KUKA KRL program: f1_Kuka_APT215T03S15.SRC

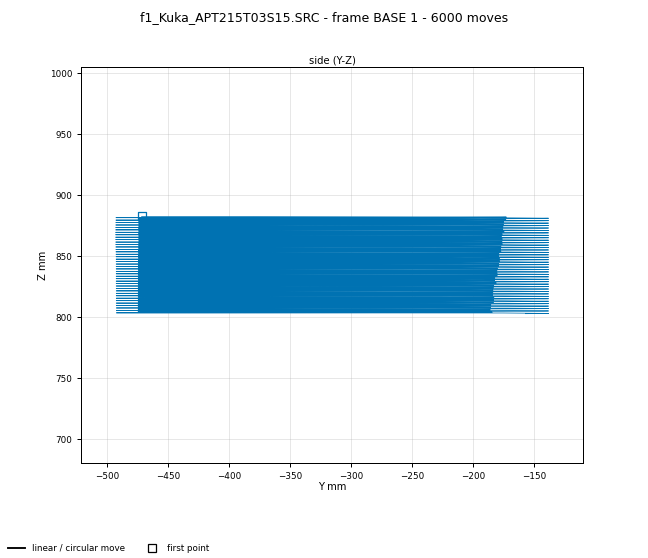
[picture p0: tool path of f1_Kuka_APT215T03S15.SRC in frame BASE 1, 6000 of 6001 moves have a stored position in this frame; points joined in program order, loops and branches not executed]
&ACCESS RVP
&REL 2
&PARAM TEMPLATE = C:\KRC\Roboter\Template\vorgabe
&PARAM EDITMASK = *
DEF f1_Kuka_APT215T03S15()


;FOLD INI;%{PE}%V3.2.0,%MKUKATPBASIS,%CINIT,%VCOMMON,%P
  ;FOLD BAS INI;%{E}%V3.2.0,%MKUKATPBASIS,%CINIT,%VINIT,%P
    GLOBAL INTERRUPT DECL 3 WHEN $STOPMESS==TRUE DO IR_STOPM ( )
    INTERRUPT ON 3
    BAS (#INITMOV,0 )
  ;ENDFOLD (BAS INI)
  ;FOLD USER INI;%{E}%V3.2.0,%MKUKATPUSER,%CINIT,%VINIT,%P
    ;Make your modifications here
  ;ENDFOLD (USER INI)
;ENDFOLD (INI)


;*** Make Null PTP Move
  PTP $pos_act

;*** Auto Load The Correct TOOL Data
  $tool=tool_data[3]

;*** Auto Load The Correct BASE Data
  $base=base_data[1]

  $ADVANCE = 5

;*** Restate Last Velocity
MMPM(30000.0)
SetRPM(6000)
LIN {X 0.010,Y -471.850,Z 882.542,A 0.000,B 0.000,C 90.000,E1 97.466} C_DIS
LIN {X -0.193,Y -470.473,Z 882.540,A 0.000,B 0.000,C 90.000,E1 97.239} C_DIS
LIN {X -0.077,Y -455.997,Z 882.527,A 0.000,B 0.000,C 90.000,E1 94.935} C_DIS
LIN {X -0.109,Y -443.986,Z 882.516,A 0.000,B 0.000,C 90.000,E1 92.865} C_DIS
LIN {X -0.078,Y -436.155,Z 882.509,A 0.000,B 0.000,C 90.000,E1 91.547} C_DIS
LIN {X -0.026,Y -426.626,Z 882.500,A 0.000,B 0.000,C 90.000,E1 89.943} C_DIS
LIN {X -0.024,Y -415.186,Z 882.489,A 0.000,B 0.000,C 90.000,E1 88.051} C_DIS
LIN {X 0.145,Y -403.849,Z 882.478,A 0.000,B 0.000,C 90.000,E1 86.102} C_DIS
LIN {X 0.181,Y -390.966,Z 882.466,A 0.000,B 0.000,C 90.000,E1 83.856} C_DIS
LIN {X -0.053,Y -379.852,Z 882.455,A 0.000,B 0.000,C 90.000,E1 81.894} C_DIS
LIN {X -0.034,Y -368.671,Z 882.444,A 0.000,B 0.000,C 90.000,E1 79.859} C_DIS
LIN {X 0.178,Y -357.598,Z 882.432,A 0.000,B 0.000,C 90.000,E1 77.757} C_DIS
LIN {X -0.125,Y -346.414,Z 882.420,A 0.000,B 0.000,C 90.000,E1 75.700} C_DIS
LIN {X 0.159,Y -333.850,Z 882.407,A 0.000,B 0.000,C 90.000,E1 73.196} C_DIS
LIN {X -0.086,Y -321.740,Z 882.393,A 0.000,B 0.000,C 90.000,E1 70.732} C_DIS
LIN {X 0.000,Y -309.964,Z 882.379,A 0.000,B 0.000,C 90.000,E1 68.156} C_DIS
LIN {X 0.018,Y -299.904,Z 882.366,A 0.000,B 0.000,C 90.000,E1 65.869} C_DIS
LIN {X -0.085,Y -289.792,Z 882.353,A 0.000,B 0.000,C 90.000,E1 63.563} C_DIS
LIN {X -0.007,Y -279.667,Z 882.340,A 0.000,B 0.000,C 90.000,E1 61.179} C_DIS
LIN {X 0.035,Y -268.308,Z 882.325,A 0.000,B 0.000,C 90.000,E1 58.408} C_DIS
LIN {X -0.117,Y -256.237,Z 882.307,A 0.000,B 0.000,C 90.000,E1 55.261} C_DIS
LIN {X -0.007,Y -245.352,Z 882.289,A 0.000,B 0.000,C 90.000,E1 51.984} C_DIS
LIN {X 0.087,Y -236.617,Z 882.272,A 0.000,B 0.000,C 90.000,E1 49.013} C_DIS
LIN {X -0.003,Y -226.592,Z 882.252,A 0.000,B 0.000,C 90.000,E1 45.283} C_DIS
LIN {X -0.070,Y -217.235,Z 882.230,A 0.000,B 0.000,C 90.000,E1 41.472} C_DIS
LIN {X 0.094,Y -208.562,Z 882.209,A 0.000,B 0.000,C 90.000,E1 37.523} C_DIS
LIN {X -0.113,Y -202.133,Z 882.191,A 0.000,B 0.000,C 90.000,E1 34.405} C_DIS
LIN {X 0.076,Y -196.229,Z 882.173,A 0.000,B 0.000,C 90.000,E1 31.131} C_DIS
LIN {X -0.021,Y -190.898,Z 882.155,A 0.000,B 0.000,C 90.000,E1 27.897} C_DIS
LIN {X -0.002,Y -186.219,Z 882.137,A 0.000,B 0.000,C 90.000,E1 24.591} C_DIS
LIN {X -0.079,Y -182.268,Z 882.118,A 0.000,B 0.000,C 90.000,E1 21.280} C_DIS
LIN {X 0.019,Y -178.306,Z 882.095,A 0.000,B 0.000,C 90.000,E1 17.040} C_DIS
LIN {X -0.012,Y -175.022,Z 882.066,A 0.000,B 0.000,C 90.000,E1 11.951} C_DIS
LIN {X -0.015,Y -172.998,Z 882.024,A 0.000,B 0.000,C 90.000,E1 4.245} C_DIS
LIN {X 0.007,Y -174.503,Z 881.974,A 0.000,B 0.000,C 90.000,E1 355.241} C_DIS
LIN {X 0.070,Y -177.369,Z 881.945,A 0.000,B 0.000,C 90.000,E1 350.095} C_DIS
LIN {X -0.017,Y -180.888,Z 881.922,A 0.000,B 0.000,C 90.000,E1 345.880} C_DIS
LIN {X 0.057,Y -184.611,Z 881.903,A 0.000,B 0.000,C 90.000,E1 342.489} C_DIS
LIN {X 0.038,Y -189.077,Z 881.884,A 0.000,B 0.000,C 90.000,E1 339.156} C_DIS
LIN {X -0.021,Y -194.301,Z 881.866,A 0.000,B 0.000,C 90.000,E1 335.869} C_DIS
LIN {X 0.062,Y -201.598,Z 881.843,A 0.000,B 0.000,C 90.000,E1 331.769} C_DIS
LIN {X -0.041,Y -209.434,Z 881.821,A 0.000,B 0.000,C 90.000,E1 327.788} C_DIS
LIN {X 0.024,Y -218.033,Z 881.799,A 0.000,B 0.000,C 90.000,E1 323.829} C_DIS
LIN {X 0.049,Y -225.580,Z 881.782,A 0.000,B 0.000,C 90.000,E1 320.723} C_DIS
LIN {X 0.044,Y -233.817,Z 881.765,A 0.000,B 0.000,C 90.000,E1 317.676} C_DIS
LIN {X 0.081,Y -243.078,Z 881.748,A 0.000,B 0.000,C 90.000,E1 314.676} C_DIS
LIN {X 0.028,Y -254.595,Z 881.730,A 0.000,B 0.000,C 90.000,E1 311.391} C_DIS
LIN {X -0.008,Y -267.268,Z 881.712,A 0.000,B 0.000,C 90.000,E1 308.177} C_DIS
LIN {X 0.040,Y -281.099,Z 881.695,A 0.000,B 0.000,C 90.000,E1 305.025} C_DIS
LIN {X -0.167,Y -296.298,Z 881.678,A 0.000,B 0.000,C 90.000,E1 302.005} C_DIS
LIN {X -0.039,Y -311.051,Z 881.663,A 0.000,B 0.000,C 90.000,E1 299.333} C_DIS
LIN {X 0.005,Y -323.057,Z 881.652,A 0.000,B 0.000,C 90.000,E1 297.385} C_DIS
LIN {X 0.118,Y -338.511,Z 881.640,A 0.000,B 0.000,C 90.000,E1 295.155} C_DIS
LIN {X 0.107,Y -357.539,Z 881.626,A 0.000,B 0.000,C 90.000,E1 292.717} C_DIS
LIN {X 0.020,Y -380.471,Z 881.612,A 0.000,B 0.000,C 90.000,E1 290.066} C_DIS
LIN {X -0.081,Y -403.987,Z 881.598,A 0.000,B 0.000,C 90.000,E1 287.583} C_DIS
LIN {X -0.193,Y -416.845,Z 881.590,A 0.000,B 0.000,C 90.000,E1 286.260} C_DIS
LIN {X -0.043,Y -429.200,Z 881.583,A 0.000,B 0.000,C 90.000,E1 284.898} C_DIS
LIN {X -0.037,Y -438.799,Z 881.577,A 0.000,B 0.000,C 90.000,E1 283.828} C_DIS
LIN {X 0.178,Y -450.162,Z 881.569,A 0.000,B 0.000,C 90.000,E1 282.479} C_DIS
LIN {X 0.044,Y -456.611,Z 881.565,A 0.000,B 0.000,C 90.000,E1 281.715} C_DIS
LIN {X 0.242,Y -464.630,Z 881.559,A 0.000,B 0.000,C 90.000,E1 280.658} C_DIS
LIN {X -0.013,Y -472.017,Z 881.554,A 0.000,B 0.000,C 90.000,E1 279.670} C_DIS
LIN {X -0.192,Y -478.710,Z 881.548,A 0.000,B 0.000,C 90.000,E1 278.681} C_DIS
LIN {X -0.246,Y -482.946,Z 881.544,A 0.000,B 0.000,C 90.000,E1 277.936} C_DIS
LIN {X -0.189,Y -486.486,Z 881.540,A 0.000,B 0.000,C 90.000,E1 277.182} C_DIS
LIN {X -0.107,Y -489.356,Z 881.536,A 0.000,B 0.000,C 90.000,E1 276.429} C_DIS
LIN {X 0.102,Y -490.795,Z 881.533,A 0.000,B 0.000,C 90.000,E1 275.910} C_DIS
LIN {X -0.169,Y -491.904,Z 881.530,A 0.000,B 0.000,C 90.000,E1 275.448} C_DIS
LIN {X 0.014,Y -492.581,Z 881.527,A 0.000,B 0.000,C 90.000,E1 274.935} C_DIS
LIN {X -0.244,Y -492.872,Z 881.525,A 0.000,B 0.000,C 90.000,E1 274.473} C_DIS
LIN {X -0.009,Y -492.764,Z 881.522,A 0.000,B 0.000,C 90.000,E1 273.955} C_DIS
LIN {X 0.195,Y -492.202,Z 881.519,A 0.000,B 0.000,C 90.000,E1 273.440} C_DIS
LIN {X -0.063,Y -491.234,Z 881.517,A 0.000,B 0.000,C 90.000,E1 272.980} C_DIS
LIN {X 0.140,Y -489.732,Z 881.514,A 0.000,B 0.000,C 90.000,E1 272.465} C_DIS
LIN {X -0.149,Y -487.740,Z 881.511,A 0.000,B 0.000,C 90.000,E1 272.007} C_DIS
LIN {X 0.058,Y -485.217,Z 881.508,A 0.000,B 0.000,C 90.000,E1 271.489} C_DIS
LIN {X 0.229,Y -481.976,Z 881.506,A 0.000,B 0.000,C 90.000,E1 270.974} C_DIS
LIN {X -0.096,Y -477.977,Z 881.503,A 0.000,B 0.000,C 90.000,E1 270.516} C_DIS
LIN {X 0.039,Y -473.005,Z 881.500,A 0.000,B 0.000,C 90.000,E1 270.000} C_DIS
LIN {X -0.168,Y -467.225,Z 881.497,A 0.000,B 0.000,C 90.000,E1 269.542} C_DIS
LIN {X 0.073,Y -461.050,Z 881.495,A 0.000,B 0.000,C 90.000,E1 269.083} C_DIS
LIN {X -0.184,Y -454.316,Z 881.493,A 0.000,B 0.000,C 90.000,E1 268.740} C_DIS
LIN {X 0.053,Y -447.342,Z 881.491,A 0.000,B 0.000,C 90.000,E1 268.396} C_DIS
LIN {X -0.151,Y -439.936,Z 881.490,A 0.000,B 0.000,C 90.000,E1 268.165} C_DIS
LIN {X 0.051,Y -432.196,Z 881.489,A 0.000,B 0.000,C 90.000,E1 267.936} C_DIS
LIN {X 0.202,Y -424.431,Z 881.488,A 0.000,B 0.000,C 90.000,E1 267.764} C_DIS
LIN {X -0.029,Y -417.358,Z 881.487,A 0.000,B 0.000,C 90.000,E1 267.707} C_DIS
LIN {X 0.050,Y -409.094,Z 881.487,A 0.000,B 0.000,C 90.000,E1 267.650} C_DIS
LIN {X -0.005,Y -181.071,Z 881.487,A 0.000,B 0.000,C 90.000,E1 267.650} C_DIS
LIN {X 0.042,Y -180.878,Z 881.473,A 0.000,B 0.000,C 90.000,E1 265.065} C_DIS
LIN {X -0.078,Y -178.996,Z 881.445,A 0.000,B 0.000,C 90.000,E1 260.038} C_DIS
LIN {X 0.016,Y -178.582,Z 881.440,A 0.000,B 0.000,C 90.000,E1 259.162} C_DIS
LIN {X -0.090,Y -175.636,Z 881.411,A 0.000,B 0.000,C 90.000,E1 254.102} C_DIS
LIN {X -0.024,Y -172.355,Z 881.388,A 0.000,B 0.000,C 90.000,E1 249.806} C_DIS
LIN {X -0.069,Y -171.140,Z 881.378,A 0.000,B 0.000,C 90.000,E1 248.103} C_DIS
LIN {X -0.024,Y -167.444,Z 881.354,A 0.000,B 0.000,C 90.000,E1 243.768} C_DIS
LIN {X 0.058,Y -166.840,Z 881.349,A 0.000,B 0.000,C 90.000,E1 242.871} C_DIS
LIN {X -0.025,Y -162.823,Z 881.325,A 0.000,B 0.000,C 90.000,E1 238.535} C_DIS
LIN {X 0.039,Y -161.509,Z 881.315,A 0.000,B 0.000,C 90.000,E1 236.755} C_DIS
LIN {X -0.008,Y -157.507,Z 881.291,A 0.000,B 0.000,C 90.000,E1 232.351} C_DIS
LIN {X 0.026,Y -155.529,Z 881.276,A 0.000,B 0.000,C 90.000,E1 229.666} C_DIS
LIN {X 0.075,Y -151.826,Z 881.251,A 0.000,B 0.000,C 90.000,E1 225.162} C_DIS
LIN {X 0.087,Y -150.040,Z 881.236,A 0.000,B 0.000,C 90.000,E1 222.447} C_DIS
LIN {X 0.001,Y -146.857,Z 881.211,A 0.000,B 0.000,C 90.000,E1 217.935} C_DIS
LIN {X 0.019,Y -145.441,Z 881.195,A 0.000,B 0.000,C 90.000,E1 215.185} C_DIS
LIN {X 0.014,Y -142.862,Z 881.170,A 0.000,B 0.000,C 90.000,E1 210.590} C_DIS
LIN {X 0.066,Y -141.478,Z 881.149,A 0.000,B 0.000,C 90.000,E1 206.873} C_DIS
LIN {X -0.074,Y -139.380,Z 881.113,A 0.000,B 0.000,C 90.000,E1 200.429} C_DIS
LIN {X 0.047,Y -138.834,Z 881.098,A 0.000,B 0.000,C 90.000,E1 197.583} C_DIS
LIN {X -0.025,Y -138.354,Z 881.056,A 0.000,B 0.000,C 90.000,E1 190.141} C_DIS
LIN {X -0.030,Y -139.524,Z 881.004,A 0.000,B 0.000,C 90.000,E1 180.802} C_DIS
LIN {X 0.063,Y -141.193,Z 880.973,A 0.000,B 0.000,C 90.000,E1 175.179} C_DIS
LIN {X 0.022,Y -142.570,Z 880.958,A 0.000,B 0.000,C 90.000,E1 172.413} C_DIS
LIN {X -0.023,Y -144.858,Z 880.932,A 0.000,B 0.000,C 90.000,E1 167.813} C_DIS
LIN {X -0.068,Y -147.484,Z 880.912,A 0.000,B 0.000,C 90.000,E1 164.157} C_DIS
LIN {X -0.042,Y -150.071,Z 880.892,A 0.000,B 0.000,C 90.000,E1 160.496} C_DIS
LIN {X -0.039,Y -153.420,Z 880.871,A 0.000,B 0.000,C 90.000,E1 156.869} C_DIS
LIN {X 0.010,Y -156.840,Z 880.851,A 0.000,B 0.000,C 90.000,E1 153.256} C_DIS
LIN {X 0.081,Y -160.920,Z 880.832,A 0.000,B 0.000,C 90.000,E1 149.665} C_DIS
LIN {X 0.026,Y -163.045,Z 880.822,A 0.000,B 0.000,C 90.000,E1 147.916} C_DIS
LIN {X 0.030,Y -167.437,Z 880.802,A 0.000,B 0.000,C 90.000,E1 144.402} C_DIS
LIN {X -0.060,Y -171.275,Z 880.788,A 0.000,B 0.000,C 90.000,E1 141.823} C_DIS
LIN {X -0.022,Y -176.168,Z 880.769,A 0.000,B 0.000,C 90.000,E1 138.366} C_DIS
LIN {X -0.024,Y -180.440,Z 880.754,A 0.000,B 0.000,C 90.000,E1 135.810} C_DIS
LIN {X -0.048,Y -185.845,Z 880.736,A 0.000,B 0.000,C 90.000,E1 132.447} C_DIS
LIN {X 0.005,Y -190.467,Z 880.722,A 0.000,B 0.000,C 90.000,E1 129.930} C_DIS
LIN {X -0.053,Y -193.245,Z 880.713,A 0.000,B 0.000,C 90.000,E1 128.302} C_DIS
LIN {X 0.114,Y -294.589,Z 880.713,A 0.000,B 0.000,C 90.000,E1 128.257} C_DIS
LIN {X -0.011,Y -298.435,Z 880.712,A 0.000,B 0.000,C 90.000,E1 128.177} C_DIS
LIN {X 0.067,Y -301.502,Z 880.711,A 0.000,B 0.000,C 90.000,E1 127.971} C_DIS
LIN {X 0.003,Y -305.177,Z 880.709,A 0.000,B 0.000,C 90.000,E1 127.604} C_DIS
LIN {X -0.028,Y -308.676,Z 880.706,A 0.000,B 0.000,C 90.000,E1 127.030} C_DIS
LIN {X -0.066,Y -310.063,Z 880.704,A 0.000,B 0.000,C 90.000,E1 126.710} C_DIS
LIN {X -0.025,Y -313.058,Z 880.698,A 0.000,B 0.000,C 90.000,E1 125.724} C_DIS
LIN {X 0.026,Y -323.493,Z 880.681,A 0.000,B 0.000,C 90.000,E1 122.498} C_DIS
LIN {X -0.040,Y -334.226,Z 880.665,A 0.000,B 0.000,C 90.000,E1 119.667} C_DIS
LIN {X -0.012,Y -346.336,Z 880.649,A 0.000,B 0.000,C 90.000,E1 116.873} C_DIS
LIN {X 0.053,Y -359.926,Z 880.634,A 0.000,B 0.000,C 90.000,E1 114.131} C_DIS
LIN {X -0.037,Y -373.349,Z 880.621,A 0.000,B 0.000,C 90.000,E1 111.770} C_DIS
LIN {X -0.066,Y -388.134,Z 880.608,A 0.000,B 0.000,C 90.000,E1 109.450} C_DIS
LIN {X 0.029,Y -404.388,Z 880.595,A 0.000,B 0.000,C 90.000,E1 107.166} C_DIS
LIN {X 0.029,Y -422.226,Z 880.583,A 0.000,B 0.000,C 90.000,E1 104.954} C_DIS
LIN {X -0.091,Y -441.673,Z 880.571,A 0.000,B 0.000,C 90.000,E1 102.827} C_DIS
LIN {X -0.072,Y -461.927,Z 880.560,A 0.000,B 0.000,C 90.000,E1 100.838} C_DIS
LIN {X -0.063,Y -467.060,Z 880.558,A 0.000,B 0.000,C 90.000,E1 100.366} C_DIS
LIN {X -0.122,Y -469.152,Z 880.556,A 0.000,B 0.000,C 90.000,E1 100.141} C_DIS
LIN {X 0.189,Y -470.867,Z 880.555,A 0.000,B 0.000,C 90.000,E1 99.849} C_DIS
LIN {X 0.037,Y -472.156,Z 880.553,A 0.000,B 0.000,C 90.000,E1 99.613} C_DIS
LIN {X 0.140,Y -473.756,Z 880.551,A 0.000,B 0.000,C 90.000,E1 99.095} C_DIS
LIN {X -0.144,Y -474.301,Z 880.548,A 0.000,B 0.000,C 90.000,E1 98.624} C_DIS
LIN {X -0.022,Y -473.883,Z 880.545,A 0.000,B 0.000,C 90.000,E1 98.106} C_DIS
LIN {X 0.105,Y -472.441,Z 880.542,A 0.000,B 0.000,C 90.000,E1 97.587} C_DIS
LIN {X -0.036,Y -471.263,Z 880.541,A 0.000,B 0.000,C 90.000,E1 97.352} C_DIS
LIN {X 0.122,Y -453.784,Z 880.525,A 0.000,B 0.000,C 90.000,E1 94.531} C_DIS
LIN {X -0.184,Y -443.285,Z 880.515,A 0.000,B 0.000,C 90.000,E1 92.751} C_DIS
LIN {X 0.163,Y -432.309,Z 880.505,A 0.000,B 0.000,C 90.000,E1 90.859} C_DIS
LIN {X 0.015,Y -424.286,Z 880.497,A 0.000,B 0.000,C 90.000,E1 89.542} C_DIS
LIN {X 0.054,Y -411.223,Z 880.485,A 0.000,B 0.000,C 90.000,E1 87.364} C_DIS
LIN {X -0.162,Y -398.253,Z 880.473,A 0.000,B 0.000,C 90.000,E1 85.179} C_DIS
LIN {X 0.146,Y -385.479,Z 880.461,A 0.000,B 0.000,C 90.000,E1 82.875} C_DIS
LIN {X -0.146,Y -374.324,Z 880.449,A 0.000,B 0.000,C 90.000,E1 80.905} C_DIS
LIN {X 0.098,Y -361.590,Z 880.436,A 0.000,B 0.000,C 90.000,E1 78.522} C_DIS
LIN {X -0.063,Y -352.080,Z 880.426,A 0.000,B 0.000,C 90.000,E1 76.756} C_DIS
LIN {X -0.144,Y -339.421,Z 880.413,A 0.000,B 0.000,C 90.000,E1 74.338} C_DIS
LIN {X 0.024,Y -325.599,Z 880.397,A 0.000,B 0.000,C 90.000,E1 71.511} C_DIS
LIN {X 0.166,Y -315.230,Z 880.385,A 0.000,B 0.000,C 90.000,E1 69.263} C_DIS
LIN {X 0.096,Y -302.213,Z 880.369,A 0.000,B 0.000,C 90.000,E1 66.357} C_DIS
LIN {X -0.080,Y -292.138,Z 880.356,A 0.000,B 0.000,C 90.000,E1 64.076} C_DIS
LIN {X 0.047,Y -282.052,Z 880.343,A 0.000,B 0.000,C 90.000,E1 61.691} C_DIS
LIN {X 0.014,Y -270.690,Z 880.328,A 0.000,B 0.000,C 90.000,E1 58.948} C_DIS
LIN {X -0.027,Y -257.195,Z 880.308,A 0.000,B 0.000,C 90.000,E1 55.435} C_DIS
LIN {X -0.032,Y -246.268,Z 880.290,A 0.000,B 0.000,C 90.000,E1 52.190} C_DIS
LIN {X 0.050,Y -235.395,Z 880.269,A 0.000,B 0.000,C 90.000,E1 48.485} C_DIS
LIN {X -0.079,Y -225.504,Z 880.249,A 0.000,B 0.000,C 90.000,E1 44.757} C_DIS
LIN {X -0.026,Y -216.257,Z 880.227,A 0.000,B 0.000,C 90.000,E1 40.906} C_DIS
LIN {X -0.127,Y -209.338,Z 880.210,A 0.000,B 0.000,C 90.000,E1 37.810} C_DIS
LIN {X -0.027,Y -202.848,Z 880.192,A 0.000,B 0.000,C 90.000,E1 34.612} C_DIS
LIN {X 0.010,Y -196.935,Z 880.174,A 0.000,B 0.000,C 90.000,E1 31.386} C_DIS
LIN {X -0.071,Y -191.539,Z 880.156,A 0.000,B 0.000,C 90.000,E1 28.153} C_DIS
LIN {X 0.043,Y -186.802,Z 880.138,A 0.000,B 0.000,C 90.000,E1 24.823} C_DIS
LIN {X -0.095,Y -182.794,Z 880.119,A 0.000,B 0.000,C 90.000,E1 21.535} C_DIS
LIN {X 0.080,Y -178.782,Z 880.096,A 0.000,B 0.000,C 90.000,E1 17.275} C_DIS
LIN {X 0.063,Y -175.424,Z 880.068,A 0.000,B 0.000,C 90.000,E1 12.187} C_DIS
LIN {X -0.071,Y -173.297,Z 880.025,A 0.000,B 0.000,C 90.000,E1 4.531} C_DIS
LIN {X 0.017,Y -174.836,Z 879.974,A 0.000,B 0.000,C 90.000,E1 355.241} C_DIS
LIN {X 0.093,Y -177.721,Z 879.945,A 0.000,B 0.000,C 90.000,E1 350.095} C_DIS
LIN {X 0.016,Y -181.260,Z 879.922,A 0.000,B 0.000,C 90.000,E1 345.880} C_DIS
LIN {X -0.029,Y -186.033,Z 879.898,A 0.000,B 0.000,C 90.000,E1 341.692} C_DIS
LIN {X 0.060,Y -190.719,Z 879.880,A 0.000,B 0.000,C 90.000,E1 338.337} C_DIS
LIN {X 0.046,Y -196.088,Z 879.861,A 0.000,B 0.000,C 90.000,E1 335.049} C_DIS
LIN {X 0.006,Y -203.451,Z 879.839,A 0.000,B 0.000,C 90.000,E1 331.001} C_DIS
LIN {X 0.053,Y -209.729,Z 879.821,A 0.000,B 0.000,C 90.000,E1 327.788} C_DIS
LIN {X 0.003,Y -218.309,Z 879.799,A 0.000,B 0.000,C 90.000,E1 323.863} C_DIS
LIN {X -0.150,Y -225.862,Z 879.782,A 0.000,B 0.000,C 90.000,E1 320.803} C_DIS
LIN {X 0.017,Y -234.095,Z 879.765,A 0.000,B 0.000,C 90.000,E1 317.715} C_DIS
LIN {X -0.122,Y -243.332,Z 879.748,A 0.000,B 0.000,C 90.000,E1 314.757} C_DIS
LIN {X -0.008,Y -254.812,Z 879.730,A 0.000,B 0.000,C 90.000,E1 311.434} C_DIS
LIN {X -0.050,Y -267.406,Z 879.712,A 0.000,B 0.000,C 90.000,E1 308.222} C_DIS
LIN {X -0.171,Y -281.188,Z 879.695,A 0.000,B 0.000,C 90.000,E1 305.105} C_DIS
LIN {X 0.037,Y -294.547,Z 879.680,A 0.000,B 0.000,C 90.000,E1 302.339} C_DIS
LIN {X 0.128,Y -309.056,Z 879.665,A 0.000,B 0.000,C 90.000,E1 299.667} C_DIS
LIN {X -0.074,Y -322.902,Z 879.652,A 0.000,B 0.000,C 90.000,E1 297.436} C_DIS
LIN {X 0.026,Y -338.293,Z 879.640,A 0.000,B 0.000,C 90.000,E1 295.207} C_DIS
LIN {X 0.021,Y -359.692,Z 879.625,A 0.000,B 0.000,C 90.000,E1 292.461} C_DIS
LIN {X 0.155,Y -382.405,Z 879.610,A 0.000,B 0.000,C 90.000,E1 289.812} C_DIS
LIN {X -0.110,Y -403.327,Z 879.598,A 0.000,B 0.000,C 90.000,E1 287.638} C_DIS
LIN {X 0.178,Y -416.194,Z 879.590,A 0.000,B 0.000,C 90.000,E1 286.260} C_DIS
LIN {X 0.181,Y -426.104,Z 879.585,A 0.000,B 0.000,C 90.000,E1 285.190} C_DIS
LIN {X 0.043,Y -438.088,Z 879.577,A 0.000,B 0.000,C 90.000,E1 283.883} C_DIS
LIN {X -0.192,Y -449.527,Z 879.570,A 0.000,B 0.000,C 90.000,E1 282.591} C_DIS
LIN {X -0.082,Y -458.102,Z 879.564,A 0.000,B 0.000,C 90.000,E1 281.535} C_DIS
LIN {X 0.043,Y -465.993,Z 879.558,A 0.000,B 0.000,C 90.000,E1 280.489} C_DIS
LIN {X -0.195,Y -473.265,Z 879.553,A 0.000,B 0.000,C 90.000,E1 279.500} C_DIS
LIN {X -0.222,Y -478.287,Z 879.548,A 0.000,B 0.000,C 90.000,E1 278.746} C_DIS
LIN {X -0.208,Y -482.601,Z 879.544,A 0.000,B 0.000,C 90.000,E1 277.992} C_DIS
LIN {X -0.154,Y -486.208,Z 879.540,A 0.000,B 0.000,C 90.000,E1 277.239} C_DIS
LIN {X -0.074,Y -489.141,Z 879.536,A 0.000,B 0.000,C 90.000,E1 276.486} C_DIS
LIN {X 0.131,Y -490.661,Z 879.533,A 0.000,B 0.000,C 90.000,E1 275.967} C_DIS
LIN {X -0.188,Y -491.801,Z 879.531,A 0.000,B 0.000,C 90.000,E1 275.511} C_DIS
LIN {X 0.041,Y -492.535,Z 879.528,A 0.000,B 0.000,C 90.000,E1 274.992} C_DIS
LIN {X -0.218,Y -492.923,Z 879.525,A 0.000,B 0.000,C 90.000,E1 274.531} C_DIS
LIN {X 0.017,Y -492.881,Z 879.522,A 0.000,B 0.000,C 90.000,E1 274.012} C_DIS
LIN {X 0.220,Y -492.416,Z 879.520,A 0.000,B 0.000,C 90.000,E1 273.498} C_DIS
LIN {X -0.037,Y -491.506,Z 879.517,A 0.000,B 0.000,C 90.000,E1 273.037} C_DIS
LIN {X 0.167,Y -490.044,Z 879.514,A 0.000,B 0.000,C 90.000,E1 272.522} C_DIS
LIN {X -0.121,Y -488.181,Z 879.511,A 0.000,B 0.000,C 90.000,E1 272.064} C_DIS
LIN {X 0.087,Y -485.689,Z 879.509,A 0.000,B 0.000,C 90.000,E1 271.547} C_DIS
LIN {X -0.221,Y -482.566,Z 879.506,A 0.000,B 0.000,C 90.000,E1 271.088} C_DIS
LIN {X 0.099,Y -480.775,Z 879.505,A 0.000,B 0.000,C 90.000,E1 270.802} C_DIS
LIN {X -0.230,Y -476.492,Z 879.502,A 0.000,B 0.000,C 90.000,E1 270.344} C_DIS
LIN {X -0.023,Y -471.343,Z 879.499,A 0.000,B 0.000,C 90.000,E1 269.828} C_DIS
LIN {X -0.043,Y -465.546,Z 879.496,A 0.000,B 0.000,C 90.000,E1 269.370} C_DIS
LIN {X -0.133,Y -459.283,Z 879.494,A 0.000,B 0.000,C 90.000,E1 268.969} C_DIS
LIN {X -0.222,Y -452.559,Z 879.492,A 0.000,B 0.000,C 90.000,E1 268.625} C_DIS
LIN {X 0.157,Y -445.492,Z 879.491,A 0.000,B 0.000,C 90.000,E1 268.282} C_DIS
LIN {X 0.073,Y -438.054,Z 879.489,A 0.000,B 0.000,C 90.000,E1 268.051} C_DIS
LIN {X -0.042,Y -430.234,Z 879.488,A 0.000,B 0.000,C 90.000,E1 267.879} C_DIS
LIN {X 0.193,Y -422.137,Z 879.487,A 0.000,B 0.000,C 90.000,E1 267.707} C_DIS
LIN {X 0.011,Y -413.635,Z 879.487,A 0.000,B 0.000,C 90.000,E1 267.650} C_DIS
LIN {X -0.062,Y -411.199,Z 879.487,A 0.000,B 0.000,C 90.000,E1 267.650} C_DIS
LIN {X -0.060,Y -181.069,Z 879.487,A 0.000,B 0.000,C 90.000,E1 267.650} C_DIS
LIN {X -0.009,Y -180.875,Z 879.473,A 0.000,B 0.000,C 90.000,E1 265.065} C_DIS
LIN {X 0.047,Y -178.992,Z 879.444,A 0.000,B 0.000,C 90.000,E1 259.982} C_DIS
LIN {X 0.059,Y -177.980,Z 879.435,A 0.000,B 0.000,C 90.000,E1 258.285} C_DIS
LIN {X 0.029,Y -175.624,Z 879.411,A 0.000,B 0.000,C 90.000,E1 254.047} C_DIS
LIN {X 0.089,Y -172.345,Z 879.388,A 0.000,B 0.000,C 90.000,E1 249.752} C_DIS
LIN {X 0.067,Y -171.821,Z 879.383,A 0.000,B 0.000,C 90.000,E1 248.901} C_DIS
LIN {X -0.083,Y -170.289,Z 879.373,A 0.000,B 0.000,C 90.000,E1 247.230} C_DIS
LIN {X 0.010,Y -166.827,Z 879.349,A 0.000,B 0.000,C 90.000,E1 242.871} C_DIS
LIN {X -0.073,Y -162.810,Z 879.325,A 0.000,B 0.000,C 90.000,E1 238.535} C_DIS
LIN {X -0.009,Y -161.497,Z 879.315,A 0.000,B 0.000,C 90.000,E1 236.755} C_DIS
LIN {X -0.055,Y -157.494,Z 879.291,A 0.000,B 0.000,C 90.000,E1 232.351} C_DIS
LIN {X -0.020,Y -155.513,Z 879.276,A 0.000,B 0.000,C 90.000,E1 229.666} C_DIS
LIN {X 0.029,Y -151.814,Z 879.251,A 0.000,B 0.000,C 90.000,E1 225.162} C_DIS
LIN {X 0.042,Y -150.026,Z 879.236,A 0.000,B 0.000,C 90.000,E1 222.447} C_DIS
LIN {X -0.044,Y -146.847,Z 879.211,A 0.000,B 0.000,C 90.000,E1 217.935} C_DIS
LIN {X -0.026,Y -145.429,Z 879.195,A 0.000,B 0.000,C 90.000,E1 215.185} C_DIS
LIN {X -0.030,Y -142.853,Z 879.170,A 0.000,B 0.000,C 90.000,E1 210.590} C_DIS
LIN {X 0.023,Y -141.469,Z 879.149,A 0.000,B 0.000,C 90.000,E1 206.873} C_DIS
LIN {X 0.014,Y -139.378,Z 879.113,A 0.000,B 0.000,C 90.000,E1 200.375} C_DIS
LIN {X 0.003,Y -138.829,Z 879.098,A 0.000,B 0.000,C 90.000,E1 197.583} C_DIS
LIN {X -0.069,Y -138.353,Z 879.056,A 0.000,B 0.000,C 90.000,E1 190.141} C_DIS
LIN {X 0.066,Y -139.528,Z 879.004,A 0.000,B 0.000,C 90.000,E1 180.745} C_DIS
LIN {X 0.019,Y -141.201,Z 878.973,A 0.000,B 0.000,C 90.000,E1 175.179} C_DIS
LIN {X -0.022,Y -142.577,Z 878.958,A 0.000,B 0.000,C 90.000,E1 172.413} C_DIS
LIN {X 0.074,Y -144.869,Z 878.932,A 0.000,B 0.000,C 90.000,E1 167.757} C_DIS
LIN {X 0.028,Y -147.496,Z 878.912,A 0.000,B 0.000,C 90.000,E1 164.102} C_DIS
LIN {X -0.038,Y -150.085,Z 878.891,A 0.000,B 0.000,C 90.000,E1 160.477} C_DIS
LIN {X -0.024,Y -153.438,Z 878.871,A 0.000,B 0.000,C 90.000,E1 156.847} C_DIS
LIN {X -0.031,Y -157.801,Z 878.846,A 0.000,B 0.000,C 90.000,E1 152.359} C_DIS
LIN {X 0.002,Y -162.082,Z 878.827,A 0.000,B 0.000,C 90.000,E1 148.791} C_DIS
LIN {X 0.027,Y -166.280,Z 878.807,A 0.000,B 0.000,C 90.000,E1 145.261} C_DIS
LIN {X 0.025,Y -171.298,Z 878.788,A 0.000,B 0.000,C 90.000,E1 141.778} C_DIS
LIN {X 0.060,Y -176.193,Z 878.769,A 0.000,B 0.000,C 90.000,E1 138.324} C_DIS
LIN {X -0.075,Y -180.468,Z 878.754,A 0.000,B 0.000,C 90.000,E1 135.810} C_DIS
LIN {X -0.100,Y -185.872,Z 878.736,A 0.000,B 0.000,C 90.000,E1 132.447} C_DIS
LIN {X -0.048,Y -190.497,Z 878.722,A 0.000,B 0.000,C 90.000,E1 129.930} C_DIS
LIN {X -0.015,Y -193.226,Z 878.713,A 0.000,B 0.000,C 90.000,E1 128.302} C_DIS
LIN {X -0.067,Y -294.700,Z 878.713,A 0.000,B 0.000,C 90.000,E1 128.302} C_DIS
LIN {X 0.033,Y -296.174,Z 878.713,A 0.000,B 0.000,C 90.000,E1 128.257} C_DIS
LIN {X 0.147,Y -299.561,Z 878.712,A 0.000,B 0.000,C 90.000,E1 128.096} C_DIS
LIN {X -0.122,Y -302.898,Z 878.710,A 0.000,B 0.000,C 90.000,E1 127.890} C_DIS
LIN {X -0.175,Y -306.564,Z 878.708,A 0.000,B 0.000,C 90.000,E1 127.443} C_DIS
LIN {X 0.025,Y -308.408,Z 878.706,A 0.000,B 0.000,C 90.000,E1 127.076} C_DIS
LIN {X 0.043,Y -309.846,Z 878.704,A 0.000,B 0.000,C 90.000,E1 126.744} C_DIS
LIN {X 0.050,Y -311.914,Z 878.701,A 0.000,B 0.000,C 90.000,E1 126.091} C_DIS
LIN {X -0.024,Y -322.172,Z 878.683,A 0.000,B 0.000,C 90.000,E1 122.880} C_DIS
LIN {X 0.151,Y -332.733,Z 878.667,A 0.000,B 0.000,C 90.000,E1 120.001} C_DIS
LIN {X -0.161,Y -344.659,Z 878.651,A 0.000,B 0.000,C 90.000,E1 117.257} C_DIS
LIN {X -0.148,Y -358.048,Z 878.636,A 0.000,B 0.000,C 90.000,E1 114.515} C_DIS
LIN {X 0.056,Y -371.280,Z 878.623,A 0.000,B 0.000,C 90.000,E1 112.099} C_DIS
LIN {X 0.123,Y -385.859,Z 878.610,A 0.000,B 0.000,C 90.000,E1 109.758} C_DIS
LIN {X -0.091,Y -401.890,Z 878.597,A 0.000,B 0.000,C 90.000,E1 107.511} C_DIS
LIN {X 0.234,Y -419.489,Z 878.585,A 0.000,B 0.000,C 90.000,E1 105.245} C_DIS
LIN {X 0.001,Y -438.742,Z 878.573,A 0.000,B 0.000,C 90.000,E1 103.119} C_DIS
LIN {X -0.179,Y -458.914,Z 878.562,A 0.000,B 0.000,C 90.000,E1 101.130} C_DIS
LIN {X 0.239,Y -466.634,Z 878.558,A 0.000,B 0.000,C 90.000,E1 100.366} C_DIS
LIN {X 0.175,Y -468.844,Z 878.556,A 0.000,B 0.000,C 90.000,E1 100.141} C_DIS
LIN {X 0.194,Y -470.512,Z 878.555,A 0.000,B 0.000,C 90.000,E1 99.905} C_DIS
LIN {X 0.047,Y -471.889,Z 878.554,A 0.000,B 0.000,C 90.000,E1 99.670} C_DIS
LIN {X -0.103,Y -472.912,Z 878.552,A 0.000,B 0.000,C 90.000,E1 99.434} C_DIS
LIN {X 0.005,Y -474.088,Z 878.550,A 0.000,B 0.000,C 90.000,E1 98.916} C_DIS
LIN {X 0.122,Y -474.267,Z 878.547,A 0.000,B 0.000,C 90.000,E1 98.398} C_DIS
LIN {X -0.222,Y -473.476,Z 878.544,A 0.000,B 0.000,C 90.000,E1 97.936} C_DIS
LIN {X -0.031,Y -471.593,Z 878.541,A 0.000,B 0.000,C 90.000,E1 97.409} C_DIS
LIN {X 0.089,Y -468.447,Z 878.538,A 0.000,B 0.000,C 90.000,E1 96.891} C_DIS
LIN {X 0.135,Y -454.146,Z 878.526,A 0.000,B 0.000,C 90.000,E1 94.588} C_DIS
LIN {X -0.161,Y -443.655,Z 878.516,A 0.000,B 0.000,C 90.000,E1 92.808} C_DIS
LIN {X 0.033,Y -434.281,Z 878.507,A 0.000,B 0.000,C 90.000,E1 91.203} C_DIS
LIN {X 0.052,Y -424.692,Z 878.498,A 0.000,B 0.000,C 90.000,E1 89.599} C_DIS
LIN {X 0.100,Y -411.641,Z 878.486,A 0.000,B 0.000,C 90.000,E1 87.421} C_DIS
LIN {X -0.141,Y -398.646,Z 878.473,A 0.000,B 0.000,C 90.000,E1 85.241} C_DIS
LIN {X -0.183,Y -384.273,Z 878.459,A 0.000,B 0.000,C 90.000,E1 82.704} C_DIS
LIN {X -0.126,Y -373.080,Z 878.448,A 0.000,B 0.000,C 90.000,E1 80.679} C_DIS
LIN {X 0.149,Y -360.389,Z 878.435,A 0.000,B 0.000,C 90.000,E1 78.285} C_DIS
LIN {X -0.095,Y -349.324,Z 878.423,A 0.000,B 0.000,C 90.000,E1 76.228} C_DIS
LIN {X 0.066,Y -335.194,Z 878.408,A 0.000,B 0.000,C 90.000,E1 73.449} C_DIS
LIN {X -0.096,Y -321.586,Z 878.392,A 0.000,B 0.000,C 90.000,E1 70.659} C_DIS
LIN {X -0.120,Y -309.819,Z 878.378,A 0.000,B 0.000,C 90.000,E1 68.103} C_DIS
LIN {X 0.017,Y -299.798,Z 878.366,A 0.000,B 0.000,C 90.000,E1 65.793} C_DIS
LIN {X 0.048,Y -289.733,Z 878.353,A 0.000,B 0.000,C 90.000,E1 63.461} C_DIS
LIN {X 0.000,Y -279.719,Z 878.339,A 0.000,B 0.000,C 90.000,E1 61.101} C_DIS
LIN {X 0.048,Y -268.484,Z 878.324,A 0.000,B 0.000,C 90.000,E1 58.329} C_DIS
LIN {X -0.094,Y -256.500,Z 878.306,A 0.000,B 0.000,C 90.000,E1 55.182} C_DIS
LIN {X 0.025,Y -245.718,Z 878.288,A 0.000,B 0.000,C 90.000,E1 51.904} C_DIS
LIN {X -0.091,Y -234.931,Z 878.268,A 0.000,B 0.000,C 90.000,E1 48.243} C_DIS
LIN {X -0.111,Y -227.027,Z 878.251,A 0.000,B 0.000,C 90.000,E1 45.243} C_DIS
LIN {X -0.005,Y -217.714,Z 878.230,A 0.000,B 0.000,C 90.000,E1 41.391} C_DIS
LIN {X 0.066,Y -210.707,Z 878.213,A 0.000,B 0.000,C 90.000,E1 38.257} C_DIS
LIN {X -0.033,Y -202.581,Z 878.191,A 0.000,B 0.000,C 90.000,E1 34.326} C_DIS
LIN {X 0.011,Y -195.319,Z 878.168,A 0.000,B 0.000,C 90.000,E1 30.285} C_DIS
LIN {X 0.064,Y -190.119,Z 878.150,A 0.000,B 0.000,C 90.000,E1 27.001} C_DIS
LIN {X 0.061,Y -185.633,Z 878.132,A 0.000,B 0.000,C 90.000,E1 23.695} C_DIS
LIN {X -0.001,Y -181.873,Z 878.113,A 0.000,B 0.000,C 90.000,E1 20.375} C_DIS
LIN {X 0.035,Y -178.166,Z 878.090,A 0.000,B 0.000,C 90.000,E1 16.150} C_DIS
LIN {X -0.037,Y -175.179,Z 878.061,A 0.000,B 0.000,C 90.000,E1 11.074} C_DIS
LIN {X 0.080,Y -175.968,Z 877.964,A 0.000,B 0.000,C 90.000,E1 353.514} C_DIS
LIN {X -0.098,Y -179.344,Z 877.936,A 0.000,B 0.000,C 90.000,E1 348.465} C_DIS
LIN {X 0.021,Y -182.521,Z 877.917,A 0.000,B 0.000,C 90.000,E1 345.046} C_DIS
LIN {X 0.017,Y -186.410,Z 877.898,A 0.000,B 0.000,C 90.000,E1 341.692} C_DIS
LIN {X 0.046,Y -191.093,Z 877.880,A 0.000,B 0.000,C 90.000,E1 338.358} C_DIS
LIN {X -0.051,Y -197.852,Z 877.857,A 0.000,B 0.000,C 90.000,E1 334.280} C_DIS
LIN {X 0.060,Y -205.296,Z 877.835,A 0.000,B 0.000,C 90.000,E1 330.205} C_DIS
LIN {X -0.023,Y -211.689,Z 877.817,A 0.000,B 0.000,C 90.000,E1 327.041} C_DIS
LIN {X -0.066,Y -220.396,Z 877.795,A 0.000,B 0.000,C 90.000,E1 323.130} C_DIS
LIN {X 0.095,Y -229.102,Z 877.776,A 0.000,B 0.000,C 90.000,E1 319.622} C_DIS
LIN {X 0.012,Y -237.697,Z 877.759,A 0.000,B 0.000,C 90.000,E1 316.620} C_DIS
LIN {X -0.048,Y -248.516,Z 877.740,A 0.000,B 0.000,C 90.000,E1 313.299} C_DIS
LIN {X 0.070,Y -260.424,Z 877.722,A 0.000,B 0.000,C 90.000,E1 310.011} C_DIS
LIN {X -0.139,Y -273.525,Z 877.705,A 0.000,B 0.000,C 90.000,E1 306.870} C_DIS
LIN {X 0.155,Y -287.731,Z 877.687,A 0.000,B 0.000,C 90.000,E1 303.706} C_DIS
LIN {X -0.018,Y -303.427,Z 877.671,A 0.000,B 0.000,C 90.000,E1 300.718} C_DIS
LIN {X -0.007,Y -318.685,Z 877.656,A 0.000,B 0.000,C 90.000,E1 298.103} C_DIS
LIN {X 0.095,Y -329.156,Z 877.647,A 0.000,B 0.000,C 90.000,E1 296.488} C_DIS
LIN {X 0.064,Y -352.152,Z 877.630,A 0.000,B 0.000,C 90.000,E1 293.387} C_DIS
LIN {X -0.231,Y -374.544,Z 877.615,A 0.000,B 0.000,C 90.000,E1 290.737} C_DIS
LIN {X 0.210,Y -400.452,Z 877.599,A 0.000,B 0.000,C 90.000,E1 287.873} C_DIS
LIN {X 0.009,Y -413.281,Z 877.592,A 0.000,B 0.000,C 90.000,E1 286.567} C_DIS
LIN {X 0.216,Y -423.240,Z 877.586,A 0.000,B 0.000,C 90.000,E1 285.481} C_DIS
LIN {X 0.047,Y -435.340,Z 877.579,A 0.000,B 0.000,C 90.000,E1 284.175} C_DIS
LIN {X 0.213,Y -446.985,Z 877.571,A 0.000,B 0.000,C 90.000,E1 282.827} C_DIS
LIN {X -0.145,Y -455.736,Z 877.566,A 0.000,B 0.000,C 90.000,E1 281.827} C_DIS
LIN {X -0.051,Y -463.858,Z 877.560,A 0.000,B 0.000,C 90.000,E1 280.782} C_DIS
LIN {X 0.230,Y -471.269,Z 877.554,A 0.000,B 0.000,C 90.000,E1 279.726} C_DIS
LIN {X 0.181,Y -476.475,Z 877.550,A 0.000,B 0.000,C 90.000,E1 278.973} C_DIS
LIN {X 0.183,Y -481.059,Z 877.546,A 0.000,B 0.000,C 90.000,E1 278.219} C_DIS
LIN {X 0.157,Y -484.940,Z 877.542,A 0.000,B 0.000,C 90.000,E1 277.473} C_DIS
LIN {X -0.079,Y -487.157,Z 877.539,A 0.000,B 0.000,C 90.000,E1 277.004} C_DIS
LIN {X 0.119,Y -489.044,Z 877.536,A 0.000,B 0.000,C 90.000,E1 276.486} C_DIS
LIN {X -0.162,Y -490.602,Z 877.533,A 0.000,B 0.000,C 90.000,E1 276.024} C_DIS
LIN {X 0.006,Y -491.766,Z 877.531,A 0.000,B 0.000,C 90.000,E1 275.511} C_DIS
LIN {X 0.234,Y -492.542,Z 877.528,A 0.000,B 0.000,C 90.000,E1 274.992} C_DIS
LIN {X -0.024,Y -492.976,Z 877.525,A 0.000,B 0.000,C 90.000,E1 274.531} C_DIS
LIN {X 0.211,Y -492.945,Z 877.522,A 0.000,B 0.000,C 90.000,E1 274.012} C_DIS
LIN {X -0.077,Y -492.521,Z 877.520,A 0.000,B 0.000,C 90.000,E1 273.555} C_DIS
LIN {X 0.157,Y -491.619,Z 877.517,A 0.000,B 0.000,C 90.000,E1 273.037} C_DIS
LIN {X -0.130,Y -490.260,Z 877.514,A 0.000,B 0.000,C 90.000,E1 272.579} C_DIS
LIN {X 0.073,Y -488.401,Z 877.512,A 0.000,B 0.000,C 90.000,E1 272.064} C_DIS
LIN {X -0.204,Y -485.953,Z 877.509,A 0.000,B 0.000,C 90.000,E1 271.604} C_DIS
LIN {X 0.126,Y -484.559,Z 877.507,A 0.000,B 0.000,C 90.000,E1 271.318} C_DIS
LIN {X -0.187,Y -481.152,Z 877.505,A 0.000,B 0.000,C 90.000,E1 270.859} C_DIS
LIN {X -0.035,Y -476.977,Z 877.502,A 0.000,B 0.000,C 90.000,E1 270.344} C_DIS
LIN {X 0.129,Y -471.852,Z 877.499,A 0.000,B 0.000,C 90.000,E1 269.828} C_DIS
LIN {X 0.033,Y -466.114,Z 877.497,A 0.000,B 0.000,C 90.000,E1 269.370} C_DIS
LIN {X -0.085,Y -459.905,Z 877.494,A 0.000,B 0.000,C 90.000,E1 268.969} C_DIS
LIN {X -0.200,Y -453.283,Z 877.492,A 0.000,B 0.000,C 90.000,E1 268.625} C_DIS
LIN {X 0.124,Y -446.206,Z 877.491,A 0.000,B 0.000,C 90.000,E1 268.282} C_DIS
LIN {X 0.016,Y -438.793,Z 877.489,A 0.000,B 0.000,C 90.000,E1 268.051} C_DIS
LIN {X -0.121,Y -431.075,Z 877.488,A 0.000,B 0.000,C 90.000,E1 267.879} C_DIS
LIN {X 0.091,Y -422.843,Z 877.487,A 0.000,B 0.000,C 90.000,E1 267.707} C_DIS
LIN {X -0.099,Y -414.775,Z 877.487,A 0.000,B 0.000,C 90.000,E1 267.650} C_DIS
LIN {X 0.157,Y -409.737,Z 877.487,A 0.000,B 0.000,C 90.000,E1 267.593} C_DIS
LIN {X 0.035,Y -181.064,Z 877.487,A 0.000,B 0.000,C 90.000,E1 267.593} C_DIS
LIN {X -0.069,Y -180.871,Z 877.472,A 0.000,B 0.000,C 90.000,E1 265.065} C_DIS
LIN {X -0.012,Y -178.987,Z 877.444,A 0.000,B 0.000,C 90.000,E1 259.982} C_DIS
LIN {X -0.001,Y -177.967,Z 877.435,A 0.000,B 0.000,C 90.000,E1 258.285} C_DIS
LIN {X 0.018,Y -175.610,Z 877.411,A 0.000,B 0.000,C 90.000,E1 254.031} C_DIS
LIN {X 0.030,Y -172.333,Z 877.388,A 0.000,B 0.000,C 90.000,E1 249.752} C_DIS
LIN {X 0.009,Y -171.809,Z 877.383,A 0.000,B 0.000,C 90.000,E1 248.901} C_DIS
LIN {X 0.016,Y -170.271,Z 877.373,A 0.000,B 0.000,C 90.000,E1 247.177} C_DIS
LIN {X -0.048,Y -166.813,Z 877.349,A 0.000,B 0.000,C 90.000,E1 242.871} C_DIS
LIN {X 0.010,Y -162.795,Z 877.325,A 0.000,B 0.000,C 90.000,E1 238.486} C_DIS
LIN {X 0.070,Y -161.482,Z 877.315,A 0.000,B 0.000,C 90.000,E1 236.707} C_DIS
LIN {X -0.014,Y -157.477,Z 877.291,A 0.000,B 0.000,C 90.000,E1 232.316} C_DIS
LIN {X 0.042,Y -155.494,Z 877.276,A 0.000,B 0.000,C 90.000,E1 229.622} C_DIS
LIN {X -0.025,Y -151.799,Z 877.251,A 0.000,B 0.000,C 90.000,E1 225.162} C_DIS
LIN {X -0.012,Y -150.009,Z 877.236,A 0.000,B 0.000,C 90.000,E1 222.447} C_DIS
LIN {X 0.019,Y -146.835,Z 877.211,A 0.000,B 0.000,C 90.000,E1 217.890} C_DIS
LIN {X 0.006,Y -145.417,Z 877.195,A 0.000,B 0.000,C 90.000,E1 215.152} C_DIS
LIN {X 0.041,Y -142.845,Z 877.170,A 0.000,B 0.000,C 90.000,E1 210.541} C_DIS
LIN {X -0.029,Y -141.458,Z 877.149,A 0.000,B 0.000,C 90.000,E1 206.873} C_DIS
LIN {X 0.010,Y -139.375,Z 877.113,A 0.000,B 0.000,C 90.000,E1 200.355} C_DIS
LIN {X -0.048,Y -138.825,Z 877.098,A 0.000,B 0.000,C 90.000,E1 197.583} C_DIS
LIN {X 0.041,Y -138.352,Z 877.056,A 0.000,B 0.000,C 90.000,E1 190.074} C_DIS
LIN {X 0.014,Y -139.531,Z 877.004,A 0.000,B 0.000,C 90.000,E1 180.745} C_DIS
LIN {X -0.033,Y -141.210,Z 876.973,A 0.000,B 0.000,C 90.000,E1 175.179} C_DIS
LIN {X 0.068,Y -142.585,Z 876.958,A 0.000,B 0.000,C 90.000,E1 172.356} C_DIS
LIN {X 0.022,Y -144.882,Z 876.932,A 0.000,B 0.000,C 90.000,E1 167.757} C_DIS
LIN {X -0.025,Y -147.509,Z 876.912,A 0.000,B 0.000,C 90.000,E1 164.102} C_DIS
LIN {X 0.049,Y -150.102,Z 876.891,A 0.000,B 0.000,C 90.000,E1 160.423} C_DIS
LIN {X 0.062,Y -153.459,Z 876.871,A 0.000,B 0.000,C 90.000,E1 156.794} C_DIS
LIN {X -0.086,Y -157.822,Z 876.846,A 0.000,B 0.000,C 90.000,E1 152.359} C_DIS
LIN {X -0.055,Y -162.106,Z 876.826,A 0.000,B 0.000,C 90.000,E1 148.791} C_DIS
LIN {X -0.030,Y -166.307,Z 876.807,A 0.000,B 0.000,C 90.000,E1 145.261} C_DIS
LIN {X -0.034,Y -171.323,Z 876.788,A 0.000,B 0.000,C 90.000,E1 141.778} C_DIS
LIN {X 0.000,Y -176.224,Z 876.768,A 0.000,B 0.000,C 90.000,E1 138.324} C_DIS
LIN {X -0.007,Y -180.502,Z 876.754,A 0.000,B 0.000,C 90.000,E1 135.769} C_DIS
LIN {X -0.024,Y -185.906,Z 876.736,A 0.000,B 0.000,C 90.000,E1 132.405} C_DIS
LIN {X 0.036,Y -190.533,Z 876.722,A 0.000,B 0.000,C 90.000,E1 129.886} C_DIS
LIN {X 0.027,Y -193.204,Z 876.713,A 0.000,B 0.000,C 90.000,E1 128.302} C_DIS
LIN {X 0.006,Y -294.540,Z 876.713,A 0.000,B 0.000,C 90.000,E1 128.302} C_DIS
LIN {X -0.063,Y -297.188,Z 876.712,A 0.000,B 0.000,C 90.000,E1 128.257} C_DIS
LIN {X -0.172,Y -300.650,Z 876.711,A 0.000,B 0.000,C 90.000,E1 128.096} C_DIS
LIN {X 0.055,Y -304.161,Z 876.710,A 0.000,B 0.000,C 90.000,E1 127.729} C_DIS
LIN {X -0.148,Y -307.757,Z 876.707,A 0.000,B 0.000,C 90.000,E1 127.237} C_DIS
LIN {X 0.059,Y -309.320,Z 876.705,A 0.000,B 0.000,C 90.000,E1 126.870} C_DIS
LIN {X -0.168,Y -310.548,Z 876.703,A 0.000,B 0.000,C 90.000,E1 126.583} C_DIS
LIN {X -0.039,Y -321.723,Z 876.683,A 0.000,B 0.000,C 90.000,E1 123.007} C_DIS
LIN {X 0.115,Y -332.228,Z 876.667,A 0.000,B 0.000,C 90.000,E1 120.129} C_DIS
LIN {X 0.095,Y -344.090,Z 876.652,A 0.000,B 0.000,C 90.000,E1 117.334} C_DIS
LIN {X 0.105,Y -357.418,Z 876.637,A 0.000,B 0.000,C 90.000,E1 114.591} C_DIS
LIN {X 0.106,Y -370.586,Z 876.623,A 0.000,B 0.000,C 90.000,E1 112.206} C_DIS
LIN {X 0.015,Y -385.098,Z 876.610,A 0.000,B 0.000,C 90.000,E1 109.885} C_DIS
LIN {X 0.166,Y -401.057,Z 876.598,A 0.000,B 0.000,C 90.000,E1 107.583} C_DIS
LIN {X 0.088,Y -418.577,Z 876.585,A 0.000,B 0.000,C 90.000,E1 105.371} C_DIS
LIN {X -0.181,Y -437.761,Z 876.573,A 0.000,B 0.000,C 90.000,E1 103.244} C_DIS
LIN {X 0.111,Y -457.905,Z 876.562,A 0.000,B 0.000,C 90.000,E1 101.186} C_DIS
LIN {X 0.001,Y -468.033,Z 876.557,A 0.000,B 0.000,C 90.000,E1 100.254} C_DIS
LIN {X -0.048,Y -469.950,Z 876.556,A 0.000,B 0.000,C 90.000,E1 100.018} C_DIS
LIN {X -0.178,Y -471.406,Z 876.554,A 0.000,B 0.000,C 90.000,E1 99.792} C_DIS
LIN {X -0.003,Y -473.391,Z 876.551,A 0.000,B 0.000,C 90.000,E1 99.265} C_DIS
LIN {X 0.105,Y -474.251,Z 876.549,A 0.000,B 0.000,C 90.000,E1 98.746} C_DIS
LIN {X -0.174,Y -474.135,Z 876.546,A 0.000,B 0.000,C 90.000,E1 98.276} C_DIS
LIN {X -0.049,Y -473.032,Z 876.543,A 0.000,B 0.000,C 90.000,E1 97.757} C_DIS
LIN {X -0.252,Y -472.061,Z 876.542,A 0.000,B 0.000,C 90.000,E1 97.530} C_DIS
LIN {X 0.076,Y -470.751,Z 876.540,A 0.000,B 0.000,C 90.000,E1 97.239} C_DIS
LIN {X -0.004,Y -454.731,Z 876.526,A 0.000,B 0.000,C 90.000,E1 94.702} C_DIS
LIN {X 0.152,Y -444.257,Z 876.516,A 0.000,B 0.000,C 90.000,E1 92.865} C_DIS
LIN {X -0.085,Y -434.912,Z 876.507,A 0.000,B 0.000,C 90.000,E1 91.318} C_DIS
LIN {X -0.054,Y -425.333,Z 876.498,A 0.000,B 0.000,C 90.000,E1 89.714} C_DIS
LIN {X 0.012,Y -412.277,Z 876.486,A 0.000,B 0.000,C 90.000,E1 87.535} C_DIS
LIN {X -0.208,Y -399.266,Z 876.474,A 0.000,B 0.000,C 90.000,E1 85.355} C_DIS
LIN {X 0.114,Y -386.432,Z 876.461,A 0.000,B 0.000,C 90.000,E1 83.053} C_DIS
LIN {X -0.183,Y -376.862,Z 876.452,A 0.000,B 0.000,C 90.000,E1 81.376} C_DIS
LIN {X 0.136,Y -365.715,Z 876.441,A 0.000,B 0.000,C 90.000,E1 79.285} C_DIS
LIN {X -0.005,Y -354.710,Z 876.429,A 0.000,B 0.000,C 90.000,E1 77.229} C_DIS
LIN {X 0.062,Y -343.622,Z 876.417,A 0.000,B 0.000,C 90.000,E1 75.102} C_DIS
LIN {X -0.168,Y -329.729,Z 876.402,A 0.000,B 0.000,C 90.000,E1 72.362} C_DIS
LIN {X 0.067,Y -319.282,Z 876.390,A 0.000,B 0.000,C 90.000,E1 70.115} C_DIS
LIN {X -0.001,Y -306.175,Z 876.373,A 0.000,B 0.000,C 90.000,E1 67.230} C_DIS
LIN {X 0.053,Y -296.151,Z 876.361,A 0.000,B 0.000,C 90.000,E1 64.921} C_DIS
LIN {X -0.128,Y -286.148,Z 876.348,A 0.000,B 0.000,C 90.000,E1 62.615} C_DIS
LIN {X -0.054,Y -274.813,Z 876.333,A 0.000,B 0.000,C 90.000,E1 59.871} C_DIS
LIN {X 0.060,Y -262.519,Z 876.315,A 0.000,B 0.000,C 90.000,E1 56.707} C_DIS
LIN {X 0.016,Y -252.316,Z 876.299,A 0.000,B 0.000,C 90.000,E1 53.863} C_DIS
LIN {X -0.031,Y -243.139,Z 876.283,A 0.000,B 0.000,C 90.000,E1 50.964} C_DIS
LIN {X -0.003,Y -234.637,Z 876.267,A 0.000,B 0.000,C 90.000,E1 48.000} C_DIS
LIN {X -0.032,Y -226.771,Z 876.250,A 0.000,B 0.000,C 90.000,E1 45.000} C_DIS
LIN {X 0.061,Y -217.506,Z 876.229,A 0.000,B 0.000,C 90.000,E1 41.148} C_DIS
LIN {X -0.010,Y -210.508,Z 876.211,A 0.000,B 0.000,C 90.000,E1 38.051} C_DIS
LIN {X 0.058,Y -202.439,Z 876.189,A 0.000,B 0.000,C 90.000,E1 34.072} C_DIS
LIN {X 0.030,Y -195.208,Z 876.167,A 0.000,B 0.000,C 90.000,E1 30.050} C_DIS
LIN {X -0.019,Y -190.068,Z 876.149,A 0.000,B 0.000,C 90.000,E1 26.796} C_DIS
LIN {X 0.069,Y -185.612,Z 876.130,A 0.000,B 0.000,C 90.000,E1 23.462} C_DIS
LIN {X 0.076,Y -181.901,Z 876.112,A 0.000,B 0.000,C 90.000,E1 20.120} C_DIS
LIN {X 0.103,Y -178.277,Z 876.089,A 0.000,B 0.000,C 90.000,E1 15.898} C_DIS
LIN {X -0.014,Y -175.369,Z 876.060,A 0.000,B 0.000,C 90.000,E1 10.838} C_DIS
LIN {X -0.081,Y -176.295,Z 875.964,A 0.000,B 0.000,C 90.000,E1 353.571} C_DIS
LIN {X -0.073,Y -179.703,Z 875.936,A 0.000,B 0.000,C 90.000,E1 348.465} C_DIS
LIN {X 0.036,Y -183.802,Z 875.912,A 0.000,B 0.000,C 90.000,E1 344.212} C_DIS
LIN {X 0.062,Y -187.877,Z 875.894,A 0.000,B 0.000,C 90.000,E1 340.859} C_DIS
LIN {X 0.083,Y -192.742,Z 875.875,A 0.000,B 0.000,C 90.000,E1 337.539} C_DIS
LIN {X 0.043,Y -199.627,Z 875.853,A 0.000,B 0.000,C 90.000,E1 333.461} C_DIS
LIN {X -0.051,Y -207.157,Z 875.830,A 0.000,B 0.000,C 90.000,E1 329.459} C_DIS
LIN {X -0.088,Y -213.659,Z 875.813,A 0.000,B 0.000,C 90.000,E1 326.294} C_DIS
LIN {X 0.040,Y -220.684,Z 875.795,A 0.000,B 0.000,C 90.000,E1 323.130} C_DIS
LIN {X 0.039,Y -229.378,Z 875.776,A 0.000,B 0.000,C 90.000,E1 319.666} C_DIS
LIN {X -0.031,Y -237.959,Z 875.759,A 0.000,B 0.000,C 90.000,E1 316.662} C_DIS
LIN {X 0.096,Y -248.763,Z 875.741,A 0.000,B 0.000,C 90.000,E1 313.299} C_DIS
LIN {X -0.140,Y -260.619,Z 875.723,A 0.000,B 0.000,C 90.000,E1 310.092} C_DIS
LIN {X 0.032,Y -273.646,Z 875.705,A 0.000,B 0.000,C 90.000,E1 306.870} C_DIS
LIN {X -0.062,Y -287.780,Z 875.688,A 0.000,B 0.000,C 90.000,E1 303.785} C_DIS
LIN {X 0.019,Y -303.395,Z 875.671,A 0.000,B 0.000,C 90.000,E1 300.747} C_DIS
LIN {X -0.088,Y -318.574,Z 875.656,A 0.000,B 0.000,C 90.000,E1 298.153} C_DIS
LIN {X 0.006,Y -328.994,Z 875.647,A 0.000,B 0.000,C 90.000,E1 296.539} C_DIS
LIN {X -0.045,Y -351.835,Z 875.630,A 0.000,B 0.000,C 90.000,E1 293.439} C_DIS
LIN {X -0.005,Y -374.097,Z 875.615,A 0.000,B 0.000,C 90.000,E1 290.737} C_DIS
LIN {X -0.105,Y -400.186,Z 875.599,A 0.000,B 0.000,C 90.000,E1 287.928} C_DIS
LIN {X 0.034,Y -413.077,Z 875.592,A 0.000,B 0.000,C 90.000,E1 286.567} C_DIS
LIN {X 0.135,Y -423.172,Z 875.586,A 0.000,B 0.000,C 90.000,E1 285.481} C_DIS
LIN {X 0.236,Y -435.461,Z 875.579,A 0.000,B 0.000,C 90.000,E1 284.120} C_DIS
LIN {X -0.005,Y -447.073,Z 875.571,A 0.000,B 0.000,C 90.000,E1 282.827} C_DIS
LIN {X -0.177,Y -453.726,Z 875.567,A 0.000,B 0.000,C 90.000,E1 282.063} C_DIS
LIN {X -0.018,Y -462.014,Z 875.561,A 0.000,B 0.000,C 90.000,E1 281.007} C_DIS
LIN {X 0.155,Y -469.612,Z 875.555,A 0.000,B 0.000,C 90.000,E1 279.962} C_DIS
LIN {X -0.046,Y -476.614,Z 875.550,A 0.000,B 0.000,C 90.000,E1 278.973} C_DIS
LIN {X -0.045,Y -481.167,Z 875.546,A 0.000,B 0.000,C 90.000,E1 278.219} C_DIS
LIN {X -0.010,Y -485.045,Z 875.541,A 0.000,B 0.000,C 90.000,E1 277.466} C_DIS
LIN {X 0.175,Y -487.233,Z 875.539,A 0.000,B 0.000,C 90.000,E1 276.947} C_DIS
LIN {X -0.110,Y -489.128,Z 875.536,A 0.000,B 0.000,C 90.000,E1 276.486} C_DIS
LIN {X 0.095,Y -490.659,Z 875.533,A 0.000,B 0.000,C 90.000,E1 275.967} C_DIS
LIN {X -0.224,Y -491.822,Z 875.530,A 0.000,B 0.000,C 90.000,E1 275.511} C_DIS
LIN {X 0.004,Y -492.588,Z 875.528,A 0.000,B 0.000,C 90.000,E1 274.992} C_DIS
LIN {X 0.238,Y -493.017,Z 875.525,A 0.000,B 0.000,C 90.000,E1 274.473} C_DIS
LIN {X -0.018,Y -492.985,Z 875.522,A 0.000,B 0.000,C 90.000,E1 274.012} C_DIS
LIN {X 0.186,Y -492.549,Z 875.520,A 0.000,B 0.000,C 90.000,E1 273.498} C_DIS
LIN {X -0.072,Y -491.636,Z 875.517,A 0.000,B 0.000,C 90.000,E1 273.037} C_DIS
LIN {X 0.133,Y -490.305,Z 875.514,A 0.000,B 0.000,C 90.000,E1 272.522} C_DIS
LIN {X -0.154,Y -488.401,Z 875.511,A 0.000,B 0.000,C 90.000,E1 272.064} C_DIS
LIN {X 0.056,Y -485.980,Z 875.509,A 0.000,B 0.000,C 90.000,E1 271.547} C_DIS
LIN {X 0.231,Y -482.954,Z 875.506,A 0.000,B 0.000,C 90.000,E1 271.031} C_DIS
LIN {X 0.220,Y -476.985,Z 875.502,A 0.000,B 0.000,C 90.000,E1 270.286} C_DIS
LIN {X -0.095,Y -471.854,Z 875.499,A 0.000,B 0.000,C 90.000,E1 269.828} C_DIS
LIN {X -0.196,Y -466.134,Z 875.496,A 0.000,B 0.000,C 90.000,E1 269.370} C_DIS
LIN {X 0.135,Y -459.938,Z 875.494,A 0.000,B 0.000,C 90.000,E1 268.912} C_DIS
LIN {X 0.006,Y -453.306,Z 875.492,A 0.000,B 0.000,C 90.000,E1 268.568} C_DIS
LIN {X -0.095,Y -446.234,Z 875.490,A 0.000,B 0.000,C 90.000,E1 268.282} C_DIS
LIN {X -0.182,Y -438.882,Z 875.489,A 0.000,B 0.000,C 90.000,E1 268.051} C_DIS
LIN {X 0.112,Y -431.098,Z 875.488,A 0.000,B 0.000,C 90.000,E1 267.822} C_DIS
LIN {X -0.104,Y -422.777,Z 875.487,A 0.000,B 0.000,C 90.000,E1 267.707} C_DIS
LIN {X 0.132,Y -414.310,Z 875.487,A 0.000,B 0.000,C 90.000,E1 267.593} C_DIS
LIN {X 0.058,Y -411.934,Z 875.487,A 0.000,B 0.000,C 90.000,E1 267.593} C_DIS
LIN {X -0.005,Y -181.063,Z 875.487,A 0.000,B 0.000,C 90.000,E1 267.593} C_DIS
LIN {X 0.046,Y -180.867,Z 875.472,A 0.000,B 0.000,C 90.000,E1 265.008} C_DIS
LIN {X -0.077,Y -178.981,Z 875.444,A 0.000,B 0.000,C 90.000,E1 259.982} C_DIS
LIN {X -0.066,Y -177.953,Z 875.435,A 0.000,B 0.000,C 90.000,E1 258.285} C_DIS
LIN {X -0.047,Y -175.595,Z 875.411,A 0.000,B 0.000,C 90.000,E1 254.031} C_DIS
LIN {X -0.034,Y -172.319,Z 875.387,A 0.000,B 0.000,C 90.000,E1 249.752} C_DIS
LIN {X -0.054,Y -171.797,Z 875.383,A 0.000,B 0.000,C 90.000,E1 248.901} C_DIS
LIN {X -0.018,Y -169.469,Z 875.368,A 0.000,B 0.000,C 90.000,E1 246.305} C_DIS
LIN {X 0.038,Y -166.797,Z 875.349,A 0.000,B 0.000,C 90.000,E1 242.820} C_DIS
LIN {X 0.034,Y -162.777,Z 875.325,A 0.000,B 0.000,C 90.000,E1 238.456} C_DIS
LIN {X 0.009,Y -161.466,Z 875.315,A 0.000,B 0.000,C 90.000,E1 236.707} C_DIS
LIN {X 0.050,Y -157.460,Z 875.290,A 0.000,B 0.000,C 90.000,E1 232.271} C_DIS
LIN {X -0.017,Y -155.473,Z 875.276,A 0.000,B 0.000,C 90.000,E1 229.622} C_DIS
LIN {X -0.084,Y -151.784,Z 875.251,A 0.000,B 0.000,C 90.000,E1 225.162} C_DIS
LIN {X -0.071,Y -149.991,Z 875.236,A 0.000,B 0.000,C 90.000,E1 222.447} C_DIS
LIN {X -0.038,Y -146.822,Z 875.210,A 0.000,B 0.000,C 90.000,E1 217.890} C_DIS
LIN {X 0.067,Y -145.402,Z 875.195,A 0.000,B 0.000,C 90.000,E1 215.105} C_DIS
LIN {X -0.015,Y -142.834,Z 875.170,A 0.000,B 0.000,C 90.000,E1 210.541} C_DIS
LIN {X 0.041,Y -141.448,Z 875.149,A 0.000,B 0.000,C 90.000,E1 206.821} C_DIS
LIN {X -0.045,Y -139.371,Z 875.113,A 0.000,B 0.000,C 90.000,E1 200.355} C_DIS
LIN {X 0.071,Y -138.819,Z 875.097,A 0.000,B 0.000,C 90.000,E1 197.511} C_DIS
LIN {X -0.015,Y -138.353,Z 875.056,A 0.000,B 0.000,C 90.000,E1 190.074} C_DIS
LIN {X -0.042,Y -139.534,Z 875.004,A 0.000,B 0.000,C 90.000,E1 180.745} C_DIS
LIN {X 0.052,Y -141.221,Z 874.973,A 0.000,B 0.000,C 90.000,E1 175.122} C_DIS
LIN {X 0.010,Y -142.594,Z 874.958,A 0.000,B 0.000,C 90.000,E1 172.356} C_DIS
LIN {X -0.036,Y -144.896,Z 874.932,A 0.000,B 0.000,C 90.000,E1 167.757} C_DIS
LIN {X -0.083,Y -147.525,Z 874.911,A 0.000,B 0.000,C 90.000,E1 164.102} C_DIS
LIN {X -0.009,Y -150.121,Z 874.891,A 0.000,B 0.000,C 90.000,E1 160.423} C_DIS
LIN {X 0.002,Y -153.482,Z 874.871,A 0.000,B 0.000,C 90.000,E1 156.794} C_DIS
LIN {X 0.066,Y -157.846,Z 874.846,A 0.000,B 0.000,C 90.000,E1 152.281} C_DIS
LIN {X 0.022,Y -162.131,Z 874.826,A 0.000,B 0.000,C 90.000,E1 148.742} C_DIS
LIN {X 0.002,Y -166.334,Z 874.807,A 0.000,B 0.000,C 90.000,E1 145.229} C_DIS
LIN {X 0.008,Y -171.352,Z 874.787,A 0.000,B 0.000,C 90.000,E1 141.743} C_DIS
LIN {X -0.065,Y -176.256,Z 874.768,A 0.000,B 0.000,C 90.000,E1 138.324} C_DIS
LIN {X 0.055,Y -180.539,Z 874.754,A 0.000,B 0.000,C 90.000,E1 135.729} C_DIS
LIN {X 0.033,Y -185.941,Z 874.735,A 0.000,B 0.000,C 90.000,E1 132.366} C_DIS
LIN {X -0.032,Y -190.572,Z 874.722,A 0.000,B 0.000,C 90.000,E1 129.886} C_DIS
LIN {X -0.036,Y -193.175,Z 874.713,A 0.000,B 0.000,C 90.000,E1 128.338} C_DIS
LIN {X 0.092,Y -294.023,Z 874.713,A 0.000,B 0.000,C 90.000,E1 128.302} C_DIS
LIN {X 0.015,Y -297.993,Z 874.712,A 0.000,B 0.000,C 90.000,E1 128.222} C_DIS
LIN {X -0.156,Y -300.734,Z 874.711,A 0.000,B 0.000,C 90.000,E1 128.096} C_DIS
LIN {X -0.085,Y -304.438,Z 874.710,A 0.000,B 0.000,C 90.000,E1 127.729} C_DIS
LIN {X 0.065,Y -307.983,Z 874.706,A 0.000,B 0.000,C 90.000,E1 127.156} C_DIS
LIN {X -0.160,Y -309.484,Z 874.705,A 0.000,B 0.000,C 90.000,E1 126.870} C_DIS
LIN {X 0.047,Y -310.663,Z 874.703,A 0.000,B 0.000,C 90.000,E1 126.503} C_DIS
LIN {X -0.072,Y -320.749,Z 874.685,A 0.000,B 0.000,C 90.000,E1 123.293} C_DIS
LIN {X 0.062,Y -331.125,Z 874.669,A 0.000,B 0.000,C 90.000,E1 120.413} C_DIS
LIN {X -0.130,Y -342.854,Z 874.653,A 0.000,B 0.000,C 90.000,E1 117.641} C_DIS
LIN {X -0.168,Y -356.029,Z 874.638,A 0.000,B 0.000,C 90.000,E1 114.899} C_DIS
LIN {X 0.127,Y -369.057,Z 874.625,A 0.000,B 0.000,C 90.000,E1 112.461} C_DIS
LIN {X 0.136,Y -383.416,Z 874.612,A 0.000,B 0.000,C 90.000,E1 110.120} C_DIS
LIN {X -0.137,Y -399.210,Z 874.599,A 0.000,B 0.000,C 90.000,E1 107.873} C_DIS
LIN {X 0.118,Y -416.553,Z 874.587,A 0.000,B 0.000,C 90.000,E1 105.607} C_DIS
LIN {X -0.105,Y -435.555,Z 874.575,A 0.000,B 0.000,C 90.000,E1 103.467} C_DIS
LIN {X -0.069,Y -455.636,Z 874.563,A 0.000,B 0.000,C 90.000,E1 101.422} C_DIS
LIN {X -0.255,Y -465.886,Z 874.558,A 0.000,B 0.000,C 90.000,E1 100.489} C_DIS
LIN {X -0.240,Y -468.274,Z 874.557,A 0.000,B 0.000,C 90.000,E1 100.254} C_DIS
LIN {X 0.147,Y -470.154,Z 874.555,A 0.000,B 0.000,C 90.000,E1 99.962} C_DIS
LIN {X 0.071,Y -471.578,Z 874.554,A 0.000,B 0.000,C 90.000,E1 99.726} C_DIS
LIN {X 0.168,Y -473.481,Z 874.551,A 0.000,B 0.000,C 90.000,E1 99.208} C_DIS
LIN {X -0.191,Y -474.275,Z 874.548,A 0.000,B 0.000,C 90.000,E1 98.746} C_DIS
LIN {X 0.000,Y -474.097,Z 874.546,A 0.000,B 0.000,C 90.000,E1 98.219} C_DIS
LIN {X 0.125,Y -472.926,Z 874.543,A 0.000,B 0.000,C 90.000,E1 97.701} C_DIS
LIN {X -0.016,Y -471.915,Z 874.541,A 0.000,B 0.000,C 90.000,E1 97.466} C_DIS
LIN {X -0.217,Y -470.554,Z 874.540,A 0.000,B 0.000,C 90.000,E1 97.239} C_DIS
LIN {X 0.160,Y -454.539,Z 874.526,A 0.000,B 0.000,C 90.000,E1 94.645} C_DIS
LIN {X -0.133,Y -444.076,Z 874.516,A 0.000,B 0.000,C 90.000,E1 92.865} C_DIS
LIN {X 0.066,Y -434.724,Z 874.507,A 0.000,B 0.000,C 90.000,E1 91.260} C_DIS
LIN {X 0.091,Y -425.137,Z 874.498,A 0.000,B 0.000,C 90.000,E1 89.656} C_DIS
LIN {X 0.149,Y -412.074,Z 874.486,A 0.000,B 0.000,C 90.000,E1 87.478} C_DIS
LIN {X -0.082,Y -399.063,Z 874.474,A 0.000,B 0.000,C 90.000,E1 85.298} C_DIS
LIN {X -0.153,Y -386.213,Z 874.461,A 0.000,B 0.000,C 90.000,E1 83.053} C_DIS
LIN {X -0.075,Y -376.640,Z 874.452,A 0.000,B 0.000,C 90.000,E1 81.319} C_DIS
LIN {X -0.126,Y -365.528,Z 874.440,A 0.000,B 0.000,C 90.000,E1 79.285} C_DIS
LIN {X 0.083,Y -354.524,Z 874.429,A 0.000,B 0.000,C 90.000,E1 77.173} C_DIS
LIN {X 0.140,Y -343.465,Z 874.417,A 0.000,B 0.000,C 90.000,E1 75.046} C_DIS
LIN {X -0.101,Y -329.607,Z 874.402,A 0.000,B 0.000,C 90.000,E1 72.308} C_DIS
LIN {X 0.125,Y -319.168,Z 874.389,A 0.000,B 0.000,C 90.000,E1 70.061} C_DIS
LIN {X 0.047,Y -306.092,Z 874.373,A 0.000,B 0.000,C 90.000,E1 67.177} C_DIS
LIN {X -0.049,Y -296.081,Z 874.360,A 0.000,B 0.000,C 90.000,E1 64.897} C_DIS
LIN {X 0.035,Y -286.126,Z 874.347,A 0.000,B 0.000,C 90.000,E1 62.538} C_DIS
LIN {X 0.107,Y -274.860,Z 874.332,A 0.000,B 0.000,C 90.000,E1 59.793} C_DIS
LIN {X 0.128,Y -261.291,Z 874.313,A 0.000,B 0.000,C 90.000,E1 56.294} C_DIS
LIN {X -0.127,Y -250.085,Z 874.295,A 0.000,B 0.000,C 90.000,E1 53.130} C_DIS
LIN {X -0.074,Y -238.991,Z 874.275,A 0.000,B 0.000,C 90.000,E1 49.461} C_DIS
LIN {X 0.017,Y -230.879,Z 874.258,A 0.000,B 0.000,C 90.000,E1 46.458} C_DIS
LIN {X -0.089,Y -221.354,Z 874.237,A 0.000,B 0.000,C 90.000,E1 42.690} C_DIS
LIN {X 0.047,Y -214.166,Z 874.220,A 0.000,B 0.000,C 90.000,E1 39.564} C_DIS
LIN {X -0.069,Y -207.425,Z 874.202,A 0.000,B 0.000,C 90.000,E1 36.457} C_DIS
LIN {X 0.034,Y -201.156,Z 874.185,A 0.000,B 0.000,C 90.000,E1 33.245} C_DIS
LIN {X 0.091,Y -195.432,Z 874.167,A 0.000,B 0.000,C 90.000,E1 30.001} C_DIS
LIN {X 0.052,Y -190.308,Z 874.149,A 0.000,B 0.000,C 90.000,E1 26.744} C_DIS
LIN {X -0.022,Y -185.866,Z 874.130,A 0.000,B 0.000,C 90.000,E1 23.462} C_DIS
LIN {X -0.007,Y -182.126,Z 874.112,A 0.000,B 0.000,C 90.000,E1 20.120} C_DIS
LIN {X 0.028,Y -178.520,Z 874.088,A 0.000,B 0.000,C 90.000,E1 15.898} C_DIS
LIN {X -0.079,Y -175.639,Z 874.060,A 0.000,B 0.000,C 90.000,E1 10.838} C_DIS
LIN {X 0.083,Y -176.211,Z 873.969,A 0.000,B 0.000,C 90.000,E1 354.375} C_DIS
LIN {X 0.039,Y -179.390,Z 873.941,A 0.000,B 0.000,C 90.000,E1 349.285} C_DIS
LIN {X 0.092,Y -183.261,Z 873.917,A 0.000,B 0.000,C 90.000,E1 345.046} C_DIS
LIN {X -0.067,Y -188.256,Z 873.894,A 0.000,B 0.000,C 90.000,E1 340.913} C_DIS
LIN {X -0.036,Y -193.098,Z 873.875,A 0.000,B 0.000,C 90.000,E1 337.592} C_DIS
LIN {X -0.064,Y -199.955,Z 873.853,A 0.000,B 0.000,C 90.000,E1 333.512} C_DIS
LIN {X 0.035,Y -207.467,Z 873.830,A 0.000,B 0.000,C 90.000,E1 329.459} C_DIS
LIN {X -0.019,Y -215.641,Z 873.808,A 0.000,B 0.000,C 90.000,E1 325.515} C_DIS
LIN {X -0.012,Y -222.848,Z 873.791,A 0.000,B 0.000,C 90.000,E1 322.396} C_DIS
LIN {X 0.052,Y -231.712,Z 873.772,A 0.000,B 0.000,C 90.000,E1 318.933} C_DIS
LIN {X -0.138,Y -240.513,Z 873.755,A 0.000,B 0.000,C 90.000,E1 315.972} C_DIS
LIN {X -0.111,Y -250.279,Z 873.739,A 0.000,B 0.000,C 90.000,E1 313.014} C_DIS
LIN {X 0.057,Y -262.177,Z 873.721,A 0.000,B 0.000,C 90.000,E1 309.725} C_DIS
LIN {X -0.096,Y -275.275,Z 873.703,A 0.000,B 0.000,C 90.000,E1 306.583} C_DIS
LIN {X 0.086,Y -289.490,Z 873.686,A 0.000,B 0.000,C 90.000,E1 303.452} C_DIS
LIN {X -0.028,Y -305.170,Z 873.669,A 0.000,B 0.000,C 90.000,E1 300.463} C_DIS
LIN {X 0.031,Y -320.465,Z 873.655,A 0.000,B 0.000,C 90.000,E1 297.847} C_DIS
LIN {X 0.158,Y -331.015,Z 873.646,A 0.000,B 0.000,C 90.000,E1 296.232} C_DIS
LIN {X 0.049,Y -353.922,Z 873.629,A 0.000,B 0.000,C 90.000,E1 293.153} C_DIS
LIN {X 0.087,Y -378.786,Z 873.612,A 0.000,B 0.000,C 90.000,E1 290.174} C_DIS
LIN {X -0.040,Y -402.195,Z 873.598,A 0.000,B 0.000,C 90.000,E1 287.692} C_DIS
LIN {X 0.224,Y -415.062,Z 873.591,A 0.000,B 0.000,C 90.000,E1 286.315} C_DIS
LIN {X -0.052,Y -427.592,Z 873.583,A 0.000,B 0.000,C 90.000,E1 285.009} C_DIS
LIN {X 0.095,Y -439.673,Z 873.576,A 0.000,B 0.000,C 90.000,E1 283.647} C_DIS
LIN {X 0.143,Y -448.858,Z 873.570,A 0.000,B 0.000,C 90.000,E1 282.591} C_DIS
LIN {X 0.251,Y -457.473,Z 873.564,A 0.000,B 0.000,C 90.000,E1 281.535} C_DIS
LIN {X 0.087,Y -463.543,Z 873.560,A 0.000,B 0.000,C 90.000,E1 280.782} C_DIS
LIN {X -0.178,Y -471.014,Z 873.554,A 0.000,B 0.000,C 90.000,E1 279.792} C_DIS
LIN {X -0.153,Y -476.273,Z 873.550,A 0.000,B 0.000,C 90.000,E1 279.029} C_DIS
LIN {X -0.157,Y -480.880,Z 873.546,A 0.000,B 0.000,C 90.000,E1 278.276} C_DIS
LIN {X -0.189,Y -484.807,Z 873.542,A 0.000,B 0.000,C 90.000,E1 277.530} C_DIS
LIN {X 0.056,Y -487.022,Z 873.539,A 0.000,B 0.000,C 90.000,E1 277.004} C_DIS
LIN {X 0.254,Y -488.940,Z 873.536,A 0.000,B 0.000,C 90.000,E1 276.486} C_DIS
LIN {X -0.080,Y -490.504,Z 873.533,A 0.000,B 0.000,C 90.000,E1 276.030} C_DIS
LIN {X 0.140,Y -491.738,Z 873.531,A 0.000,B 0.000,C 90.000,E1 275.511} C_DIS
LIN {X -0.123,Y -492.558,Z 873.528,A 0.000,B 0.000,C 90.000,E1 275.049} C_DIS
LIN {X 0.110,Y -492.971,Z 873.525,A 0.000,B 0.000,C 90.000,E1 274.531} C_DIS
LIN {X -0.147,Y -493.046,Z 873.523,A 0.000,B 0.000,C 90.000,E1 274.069} C_DIS
LIN {X 0.056,Y -492.650,Z 873.520,A 0.000,B 0.000,C 90.000,E1 273.555} C_DIS
LIN {X -0.201,Y -491.825,Z 873.517,A 0.000,B 0.000,C 90.000,E1 273.094} C_DIS
LIN {X 0.005,Y -490.523,Z 873.514,A 0.000,B 0.000,C 90.000,E1 272.579} C_DIS
LIN {X 0.208,Y -488.721,Z 873.512,A 0.000,B 0.000,C 90.000,E1 272.064} C_DIS
LIN {X -0.068,Y -486.339,Z 873.509,A 0.000,B 0.000,C 90.000,E1 271.604} C_DIS
LIN {X 0.110,Y -483.359,Z 873.506,A 0.000,B 0.000,C 90.000,E1 271.088} C_DIS
LIN {X -0.208,Y -479.686,Z 873.503,A 0.000,B 0.000,C 90.000,E1 270.630} C_DIS
LIN {X -0.062,Y -475.209,Z 873.501,A 0.000,B 0.000,C 90.000,E1 270.115} C_DIS
LIN {X 0.057,Y -469.757,Z 873.498,A 0.000,B 0.000,C 90.000,E1 269.599} C_DIS
LIN {X 0.079,Y -466.967,Z 873.497,A 0.000,B 0.000,C 90.000,E1 269.370} C_DIS
LIN {X -0.113,Y -460.849,Z 873.494,A 0.000,B 0.000,C 90.000,E1 268.969} C_DIS
LIN {X 0.141,Y -454.246,Z 873.492,A 0.000,B 0.000,C 90.000,E1 268.568} C_DIS
LIN {X -0.054,Y -447.141,Z 873.490,A 0.000,B 0.000,C 90.000,E1 268.282} C_DIS
LIN {X -0.206,Y -439.654,Z 873.489,A 0.000,B 0.000,C 90.000,E1 268.051} C_DIS
LIN {X 0.049,Y -431.986,Z 873.488,A 0.000,B 0.000,C 90.000,E1 267.822} C_DIS
LIN {X -0.206,Y -423.623,Z 873.487,A 0.000,B 0.000,C 90.000,E1 267.707} C_DIS
LIN {X 0.023,Y -415.256,Z 873.487,A 0.000,B 0.000,C 90.000,E1 267.593} C_DIS
LIN {X -0.122,Y -410.394,Z 873.487,A 0.000,B 0.000,C 90.000,E1 267.593} C_DIS
LIN {X -0.086,Y -181.059,Z 873.486,A 0.000,B 0.000,C 90.000,E1 267.593} C_DIS
LIN {X -0.002,Y -180.863,Z 873.472,A 0.000,B 0.000,C 90.000,E1 265.008} C_DIS
LIN {X 0.052,Y -178.978,Z 873.444,A 0.000,B 0.000,C 90.000,E1 259.926} C_DIS
LIN {X 0.062,Y -177.943,Z 873.435,A 0.000,B 0.000,C 90.000,E1 258.229} C_DIS
LIN {X 0.076,Y -175.583,Z 873.411,A 0.000,B 0.000,C 90.000,E1 253.976} C_DIS
LIN {X 0.082,Y -172.309,Z 873.387,A 0.000,B 0.000,C 90.000,E1 249.699} C_DIS
LIN {X 0.059,Y -171.787,Z 873.383,A 0.000,B 0.000,C 90.000,E1 248.847} C_DIS
LIN {X -0.063,Y -169.455,Z 873.368,A 0.000,B 0.000,C 90.000,E1 246.305} C_DIS
LIN {X -0.006,Y -166.785,Z 873.349,A 0.000,B 0.000,C 90.000,E1 242.820} C_DIS
LIN {X -0.011,Y -162.764,Z 873.325,A 0.000,B 0.000,C 90.000,E1 238.456} C_DIS
LIN {X -0.035,Y -161.454,Z 873.315,A 0.000,B 0.000,C 90.000,E1 236.707} C_DIS
LIN {X 0.006,Y -157.448,Z 873.290,A 0.000,B 0.000,C 90.000,E1 232.271} C_DIS
LIN {X -0.061,Y -155.458,Z 873.276,A 0.000,B 0.000,C 90.000,E1 229.622} C_DIS
LIN {X -0.018,Y -151.773,Z 873.251,A 0.000,B 0.000,C 90.000,E1 225.121} C_DIS
LIN {X -0.002,Y -149.977,Z 873.236,A 0.000,B 0.000,C 90.000,E1 222.405} C_DIS
LIN {X 0.009,Y -146.813,Z 873.210,A 0.000,B 0.000,C 90.000,E1 217.855} C_DIS
LIN {X 0.025,Y -145.391,Z 873.195,A 0.000,B 0.000,C 90.000,E1 215.105} C_DIS
LIN {X -0.057,Y -142.827,Z 873.170,A 0.000,B 0.000,C 90.000,E1 210.541} C_DIS
LIN {X 0.000,Y -141.439,Z 873.149,A 0.000,B 0.000,C 90.000,E1 206.821} C_DIS
LIN {X 0.045,Y -139.368,Z 873.113,A 0.000,B 0.000,C 90.000,E1 200.301} C_DIS
LIN {X 0.031,Y -138.815,Z 873.097,A 0.000,B 0.000,C 90.000,E1 197.511} C_DIS
LIN {X -0.055,Y -138.352,Z 873.056,A 0.000,B 0.000,C 90.000,E1 190.074} C_DIS
LIN {X 0.058,Y -139.538,Z 873.004,A 0.000,B 0.000,C 90.000,E1 180.688} C_DIS
LIN {X 0.011,Y -141.228,Z 872.973,A 0.000,B 0.000,C 90.000,E1 175.122} C_DIS
LIN {X -0.030,Y -142.600,Z 872.957,A 0.000,B 0.000,C 90.000,E1 172.356} C_DIS
LIN {X 0.064,Y -144.906,Z 872.932,A 0.000,B 0.000,C 90.000,E1 167.701} C_DIS
LIN {X 0.017,Y -147.534,Z 872.911,A 0.000,B 0.000,C 90.000,E1 164.047} C_DIS
LIN {X -0.051,Y -150.134,Z 872.891,A 0.000,B 0.000,C 90.000,E1 160.423} C_DIS
LIN {X -0.041,Y -153.499,Z 872.871,A 0.000,B 0.000,C 90.000,E1 156.794} C_DIS
LIN {X 0.022,Y -157.864,Z 872.846,A 0.000,B 0.000,C 90.000,E1 152.281} C_DIS
LIN {X -0.022,Y -162.150,Z 872.826,A 0.000,B 0.000,C 90.000,E1 148.742} C_DIS
LIN {X 0.093,Y -166.355,Z 872.807,A 0.000,B 0.000,C 90.000,E1 145.182} C_DIS
LIN {X -0.038,Y -171.372,Z 872.787,A 0.000,B 0.000,C 90.000,E1 141.743} C_DIS
LIN {X 0.006,Y -176.280,Z 872.768,A 0.000,B 0.000,C 90.000,E1 138.286} C_DIS
LIN {X 0.006,Y -180.565,Z 872.754,A 0.000,B 0.000,C 90.000,E1 135.729} C_DIS
LIN {X -0.015,Y -185.967,Z 872.735,A 0.000,B 0.000,C 90.000,E1 132.366} C_DIS
LIN {X 0.042,Y -190.599,Z 872.721,A 0.000,B 0.000,C 90.000,E1 129.850} C_DIS
LIN {X -0.010,Y -193.162,Z 872.713,A 0.000,B 0.000,C 90.000,E1 128.338} C_DIS
LIN {X -0.051,Y -294.477,Z 872.713,A 0.000,B 0.000,C 90.000,E1 128.338} C_DIS
LIN {X 0.026,Y -295.765,Z 872.713,A 0.000,B 0.000,C 90.000,E1 128.302} C_DIS
LIN {X -0.061,Y -298.504,Z 872.712,A 0.000,B 0.000,C 90.000,E1 128.222} C_DIS
LIN {X 0.085,Y -301.837,Z 872.711,A 0.000,B 0.000,C 90.000,E1 127.971} C_DIS
LIN {X -0.113,Y -305.485,Z 872.709,A 0.000,B 0.000,C 90.000,E1 127.604} C_DIS
LIN {X -0.031,Y -307.414,Z 872.707,A 0.000,B 0.000,C 90.000,E1 127.282} C_DIS
LIN {X 0.111,Y -308.928,Z 872.705,A 0.000,B 0.000,C 90.000,E1 126.950} C_DIS
LIN {X -0.105,Y -310.208,Z 872.704,A 0.000,B 0.000,C 90.000,E1 126.664} C_DIS
LIN {X 0.099,Y -322.474,Z 872.682,A 0.000,B 0.000,C 90.000,E1 122.752} C_DIS
LIN {X -0.002,Y -333.085,Z 872.666,A 0.000,B 0.000,C 90.000,E1 119.922} C_DIS
LIN {X -0.005,Y -345.058,Z 872.651,A 0.000,B 0.000,C 90.000,E1 117.129} C_DIS
LIN {X 0.020,Y -358.508,Z 872.635,A 0.000,B 0.000,C 90.000,E1 114.387} C_DIS
LIN {X -0.104,Y -371.793,Z 872.622,A 0.000,B 0.000,C 90.000,E1 112.025} C_DIS
LIN {X -0.039,Y -386.431,Z 872.609,A 0.000,B 0.000,C 90.000,E1 109.685} C_DIS
LIN {X 0.008,Y -402.525,Z 872.597,A 0.000,B 0.000,C 90.000,E1 107.402} C_DIS
LIN {X -0.042,Y -420.192,Z 872.584,A 0.000,B 0.000,C 90.000,E1 105.190} C_DIS
LIN {X 0.169,Y -439.509,Z 872.572,A 0.000,B 0.000,C 90.000,E1 103.008} C_DIS
LIN {X 0.148,Y -459.705,Z 872.561,A 0.000,B 0.000,C 90.000,E1 101.007} C_DIS
LIN {X 0.066,Y -467.365,Z 872.557,A 0.000,B 0.000,C 90.000,E1 100.310} C_DIS
LIN {X 0.093,Y -469.383,Z 872.556,A 0.000,B 0.000,C 90.000,E1 100.074} C_DIS
LIN {X -0.140,Y -471.047,Z 872.555,A 0.000,B 0.000,C 90.000,E1 99.849} C_DIS
LIN {X 0.174,Y -472.296,Z 872.553,A 0.000,B 0.000,C 90.000,E1 99.557} C_DIS
LIN {X -0.190,Y -473.834,Z 872.550,A 0.000,B 0.000,C 90.000,E1 99.095} C_DIS
LIN {X -0.003,Y -474.327,Z 872.548,A 0.000,B 0.000,C 90.000,E1 98.568} C_DIS
LIN {X 0.119,Y -473.858,Z 872.545,A 0.000,B 0.000,C 90.000,E1 98.049} C_DIS
LIN {X -0.221,Y -472.356,Z 872.542,A 0.000,B 0.000,C 90.000,E1 97.587} C_DIS
LIN {X 0.105,Y -471.142,Z 872.541,A 0.000,B 0.000,C 90.000,E1 97.296} C_DIS
LIN {X -0.196,Y -453.640,Z 872.525,A 0.000,B 0.000,C 90.000,E1 94.531} C_DIS
LIN {X -0.055,Y -443.170,Z 872.515,A 0.000,B 0.000,C 90.000,E1 92.694} C_DIS
LIN {X 0.129,Y -433.763,Z 872.506,A 0.000,B 0.000,C 90.000,E1 91.088} C_DIS
LIN {X 0.136,Y -424.168,Z 872.497,A 0.000,B 0.000,C 90.000,E1 89.484} C_DIS
LIN {X 0.169,Y -411.094,Z 872.485,A 0.000,B 0.000,C 90.000,E1 87.306} C_DIS
LIN {X -0.129,Y -399.704,Z 872.474,A 0.000,B 0.000,C 90.000,E1 85.412} C_DIS
LIN {X -0.181,Y -386.839,Z 872.462,A 0.000,B 0.000,C 90.000,E1 83.166} C_DIS
LIN {X -0.088,Y -377.268,Z 872.452,A 0.000,B 0.000,C 90.000,E1 81.432} C_DIS
LIN {X -0.137,Y -364.586,Z 872.439,A 0.000,B 0.000,C 90.000,E1 79.106} C_DIS
LIN {X 0.057,Y -353.580,Z 872.428,A 0.000,B 0.000,C 90.000,E1 76.992} C_DIS
LIN {X 0.099,Y -342.563,Z 872.416,A 0.000,B 0.000,C 90.000,E1 74.866} C_DIS
LIN {X -0.164,Y -328.773,Z 872.401,A 0.000,B 0.000,C 90.000,E1 72.127} C_DIS
LIN {X -0.014,Y -316.864,Z 872.386,A 0.000,B 0.000,C 90.000,E1 69.571} C_DIS
LIN {X 0.067,Y -305.341,Z 872.372,A 0.000,B 0.000,C 90.000,E1 66.975} C_DIS
LIN {X 0.101,Y -293.935,Z 872.357,A 0.000,B 0.000,C 90.000,E1 64.332} C_DIS
LIN {X -0.119,Y -284.034,Z 872.344,A 0.000,B 0.000,C 90.000,E1 62.025} C_DIS
LIN {X -0.096,Y -272.858,Z 872.329,A 0.000,B 0.000,C 90.000,E1 59.282} C_DIS
LIN {X 0.005,Y -259.488,Z 872.310,A 0.000,B 0.000,C 90.000,E1 55.754} C_DIS
LIN {X -0.151,Y -248.527,Z 872.292,A 0.000,B 0.000,C 90.000,E1 52.557} C_DIS
LIN {X 0.027,Y -238.689,Z 872.273,A 0.000,B 0.000,C 90.000,E1 49.218} C_DIS
LIN {X 0.010,Y -228.662,Z 872.253,A 0.000,B 0.000,C 90.000,E1 45.486} C_DIS
LIN {X -0.010,Y -221.132,Z 872.236,A 0.000,B 0.000,C 90.000,E1 42.447} C_DIS
LIN {X -0.021,Y -213.981,Z 872.219,A 0.000,B 0.000,C 90.000,E1 39.358} C_DIS
LIN {X -0.014,Y -207.268,Z 872.201,A 0.000,B 0.000,C 90.000,E1 36.217} C_DIS
LIN {X -0.034,Y -201.025,Z 872.183,A 0.000,B 0.000,C 90.000,E1 33.038} C_DIS
LIN {X 0.021,Y -195.333,Z 872.166,A 0.000,B 0.000,C 90.000,E1 29.795} C_DIS
LIN {X -0.024,Y -190.259,Z 872.147,A 0.000,B 0.000,C 90.000,E1 26.539} C_DIS
LIN {X 0.069,Y -185.874,Z 872.129,A 0.000,B 0.000,C 90.000,E1 23.206} C_DIS
LIN {X 0.015,Y -182.173,Z 872.110,A 0.000,B 0.000,C 90.000,E1 19.885} C_DIS
LIN {X 0.057,Y -178.614,Z 872.087,A 0.000,B 0.000,C 90.000,E1 15.662} C_DIS
LIN {X -0.047,Y -175.837,Z 872.059,A 0.000,B 0.000,C 90.000,E1 10.602} C_DIS
LIN {X -0.080,Y -176.546,Z 871.969,A 0.000,B 0.000,C 90.000,E1 354.432} C_DIS
LIN {X 0.063,Y -179.753,Z 871.941,A 0.000,B 0.000,C 90.000,E1 349.285} C_DIS
LIN {X -0.048,Y -183.636,Z 871.917,A 0.000,B 0.000,C 90.000,E1 345.102} C_DIS
LIN {X -0.018,Y -188.626,Z 871.894,A 0.000,B 0.000,C 90.000,E1 340.913} C_DIS
LIN {X -0.050,Y -193.460,Z 871.876,A 0.000,B 0.000,C 90.000,E1 337.614} C_DIS
LIN {X 0.009,Y -200.282,Z 871.853,A 0.000,B 0.000,C 90.000,E1 333.512} C_DIS
LIN {X 0.016,Y -207.775,Z 871.831,A 0.000,B 0.000,C 90.000,E1 329.488} C_DIS
LIN {X 0.080,Y -215.909,Z 871.809,A 0.000,B 0.000,C 90.000,E1 325.515} C_DIS
LIN {X -0.038,Y -223.116,Z 871.791,A 0.000,B 0.000,C 90.000,E1 322.431} C_DIS
LIN {X -0.001,Y -231.960,Z 871.772,A 0.000,B 0.000,C 90.000,E1 318.976} C_DIS
LIN {X -0.005,Y -240.765,Z 871.755,A 0.000,B 0.000,C 90.000,E1 315.972} C_DIS
LIN {X 0.034,Y -250.499,Z 871.739,A 0.000,B 0.000,C 90.000,E1 313.014} C_DIS
LIN {X 0.014,Y -262.348,Z 871.721,A 0.000,B 0.000,C 90.000,E1 309.769} C_DIS
LIN {X 0.076,Y -275.375,Z 871.703,A 0.000,B 0.000,C 90.000,E1 306.583} C_DIS
LIN {X 0.027,Y -289.537,Z 871.686,A 0.000,B 0.000,C 90.000,E1 303.499} C_DIS
LIN {X 0.165,Y -305.123,Z 871.669,A 0.000,B 0.000,C 90.000,E1 300.463} C_DIS
LIN {X -0.051,Y -320.346,Z 871.655,A 0.000,B 0.000,C 90.000,E1 297.897} C_DIS
LIN {X 0.026,Y -333.039,Z 871.644,A 0.000,B 0.000,C 90.000,E1 295.976} C_DIS
LIN {X -0.030,Y -355.975,Z 871.627,A 0.000,B 0.000,C 90.000,E1 292.898} C_DIS
LIN {X -0.030,Y -380.906,Z 871.611,A 0.000,B 0.000,C 90.000,E1 289.939} C_DIS
LIN {X 0.147,Y -401.751,Z 871.598,A 0.000,B 0.000,C 90.000,E1 287.692} C_DIS
LIN {X 0.088,Y -414.389,Z 871.591,A 0.000,B 0.000,C 90.000,E1 286.386} C_DIS
LIN {X 0.009,Y -426.868,Z 871.584,A 0.000,B 0.000,C 90.000,E1 285.064} C_DIS
LIN {X -0.141,Y -436.590,Z 871.578,A 0.000,B 0.000,C 90.000,E1 284.008} C_DIS
LIN {X -0.032,Y -445.930,Z 871.572,A 0.000,B 0.000,C 90.000,E1 282.939} C_DIS
LIN {X 0.034,Y -454.762,Z 871.566,A 0.000,B 0.000,C 90.000,E1 281.883} C_DIS
LIN {X 0.118,Y -462.975,Z 871.560,A 0.000,B 0.000,C 90.000,E1 280.838} C_DIS
LIN {X -0.154,Y -470.528,Z 871.555,A 0.000,B 0.000,C 90.000,E1 279.849} C_DIS
LIN {X -0.210,Y -475.835,Z 871.550,A 0.000,B 0.000,C 90.000,E1 279.095} C_DIS
LIN {X -0.213,Y -480.496,Z 871.546,A 0.000,B 0.000,C 90.000,E1 278.341} C_DIS
LIN {X -0.180,Y -484.495,Z 871.542,A 0.000,B 0.000,C 90.000,E1 277.587} C_DIS
LIN {X 0.003,Y -486.754,Z 871.539,A 0.000,B 0.000,C 90.000,E1 277.068} C_DIS
LIN {X 0.203,Y -488.688,Z 871.536,A 0.000,B 0.000,C 90.000,E1 276.549} C_DIS
LIN {X -0.077,Y -490.299,Z 871.534,A 0.000,B 0.000,C 90.000,E1 276.087} C_DIS
LIN {X 0.141,Y -491.591,Z 871.531,A 0.000,B 0.000,C 90.000,E1 275.568} C_DIS
LIN {X -0.124,Y -492.482,Z 871.528,A 0.000,B 0.000,C 90.000,E1 275.106} C_DIS
LIN {X 0.108,Y -492.981,Z 871.526,A 0.000,B 0.000,C 90.000,E1 274.588} C_DIS
LIN {X -0.185,Y -493.097,Z 871.523,A 0.000,B 0.000,C 90.000,E1 274.131} C_DIS
LIN {X 0.053,Y -492.802,Z 871.520,A 0.000,B 0.000,C 90.000,E1 273.612} C_DIS
LIN {X -0.204,Y -492.020,Z 871.517,A 0.000,B 0.000,C 90.000,E1 273.151} C_DIS
LIN {X 0.003,Y -490.767,Z 871.515,A 0.000,B 0.000,C 90.000,E1 272.636} C_DIS
LIN {X 0.206,Y -489.008,Z 871.512,A 0.000,B 0.000,C 90.000,E1 272.121} C_DIS
LIN {X -0.068,Y -486.750,Z 871.509,A 0.000,B 0.000,C 90.000,E1 271.661} C_DIS
LIN {X 0.111,Y -483.873,Z 871.506,A 0.000,B 0.000,C 90.000,E1 271.146} C_DIS
LIN {X -0.204,Y -480.375,Z 871.504,A 0.000,B 0.000,C 90.000,E1 270.688} C_DIS
LIN {X -0.055,Y -476.032,Z 871.501,A 0.000,B 0.000,C 90.000,E1 270.172} C_DIS
LIN {X 0.069,Y -470.786,Z 871.498,A 0.000,B 0.000,C 90.000,E1 269.656} C_DIS
LIN {X 0.004,Y -464.878,Z 871.496,A 0.000,B 0.000,C 90.000,E1 269.198} C_DIS
LIN {X 0.195,Y -461.954,Z 871.494,A 0.000,B 0.000,C 90.000,E1 268.969} C_DIS
LIN {X -0.087,Y -455.381,Z 871.492,A 0.000,B 0.000,C 90.000,E1 268.625} C_DIS
LIN {X 0.122,Y -448.461,Z 871.491,A 0.000,B 0.000,C 90.000,E1 268.282} C_DIS
LIN {X -0.103,Y -441.032,Z 871.489,A 0.000,B 0.000,C 90.000,E1 268.051} C_DIS
LIN {X 0.072,Y -433.246,Z 871.488,A 0.000,B 0.000,C 90.000,E1 267.822} C_DIS
LIN {X 0.179,Y -424.998,Z 871.487,A 0.000,B 0.000,C 90.000,E1 267.650} C_DIS
LIN {X 0.105,Y -419.084,Z 871.487,A 0.000,B 0.000,C 90.000,E1 267.593} C_DIS
LIN {X 0.140,Y -410.200,Z 871.486,A 0.000,B 0.000,C 90.000,E1 267.535} C_DIS
LIN {X 0.029,Y -181.056,Z 871.486,A 0.000,B 0.000,C 90.000,E1 267.535} C_DIS
LIN {X -0.039,Y -180.860,Z 871.472,A 0.000,B 0.000,C 90.000,E1 265.008} C_DIS
LIN {X 0.015,Y -178.974,Z 871.444,A 0.000,B 0.000,C 90.000,E1 259.926} C_DIS
LIN {X 0.025,Y -177.935,Z 871.435,A 0.000,B 0.000,C 90.000,E1 258.229} C_DIS
LIN {X 0.039,Y -175.574,Z 871.411,A 0.000,B 0.000,C 90.000,E1 253.976} C_DIS
LIN {X 0.046,Y -172.302,Z 871.387,A 0.000,B 0.000,C 90.000,E1 249.699} C_DIS
LIN {X 0.024,Y -171.780,Z 871.383,A 0.000,B 0.000,C 90.000,E1 248.847} C_DIS
LIN {X -0.004,Y -168.711,Z 871.363,A 0.000,B 0.000,C 90.000,E1 245.409} C_DIS
LIN {X 0.034,Y -166.775,Z 871.349,A 0.000,B 0.000,C 90.000,E1 242.794} C_DIS
LIN {X -0.046,Y -162.755,Z 871.325,A 0.000,B 0.000,C 90.000,E1 238.456} C_DIS
LIN {X -0.069,Y -161.445,Z 871.315,A 0.000,B 0.000,C 90.000,E1 236.707} C_DIS
LIN {X -0.027,Y -157.438,Z 871.290,A 0.000,B 0.000,C 90.000,E1 232.271} C_DIS
LIN {X 0.006,Y -155.446,Z 871.276,A 0.000,B 0.000,C 90.000,E1 229.585} C_DIS
LIN {X 0.055,Y -151.764,Z 871.251,A 0.000,B 0.000,C 90.000,E1 225.081} C_DIS
LIN {X 0.066,Y -149.967,Z 871.236,A 0.000,B 0.000,C 90.000,E1 222.366} C_DIS
LIN {X -0.023,Y -146.805,Z 871.210,A 0.000,B 0.000,C 90.000,E1 217.855} C_DIS
LIN {X -0.006,Y -145.382,Z 871.195,A 0.000,B 0.000,C 90.000,E1 215.105} C_DIS
LIN {X -0.015,Y -142.441,Z 871.164,A 0.000,B 0.000,C 90.000,E1 209.589} C_DIS
LIN {X 0.032,Y -141.433,Z 871.149,A 0.000,B 0.000,C 90.000,E1 206.796} C_DIS
LIN {X 0.014,Y -139.366,Z 871.113,A 0.000,B 0.000,C 90.000,E1 200.301} C_DIS
LIN {X 0.000,Y -138.812,Z 871.097,A 0.000,B 0.000,C 90.000,E1 197.511} C_DIS
LIN {X 0.050,Y -138.351,Z 871.056,A 0.000,B 0.000,C 90.000,E1 190.018} C_DIS
LIN {X 0.026,Y -139.539,Z 871.004,A 0.000,B 0.000,C 90.000,E1 180.688} C_DIS
LIN {X -0.021,Y -141.233,Z 870.973,A 0.000,B 0.000,C 90.000,E1 175.122} C_DIS
LIN {X -0.063,Y -142.605,Z 870.957,A 0.000,B 0.000,C 90.000,E1 172.356} C_DIS
LIN {X 0.032,Y -144.914,Z 870.932,A 0.000,B 0.000,C 90.000,E1 167.701} C_DIS
LIN {X 0.025,Y -147.543,Z 870.911,A 0.000,B 0.000,C 90.000,E1 164.031} C_DIS
LIN {X 0.057,Y -150.144,Z 870.891,A 0.000,B 0.000,C 90.000,E1 160.369} C_DIS
LIN {X -0.074,Y -153.512,Z 870.871,A 0.000,B 0.000,C 90.000,E1 156.794} C_DIS
LIN {X -0.011,Y -157.877,Z 870.846,A 0.000,B 0.000,C 90.000,E1 152.281} C_DIS
LIN {X -0.057,Y -162.164,Z 870.826,A 0.000,B 0.000,C 90.000,E1 148.742} C_DIS
LIN {X 0.057,Y -166.371,Z 870.807,A 0.000,B 0.000,C 90.000,E1 145.182} C_DIS
LIN {X 0.060,Y -171.388,Z 870.787,A 0.000,B 0.000,C 90.000,E1 141.698} C_DIS
LIN {X 0.100,Y -176.299,Z 870.768,A 0.000,B 0.000,C 90.000,E1 138.243} C_DIS
LIN {X -0.031,Y -180.586,Z 870.754,A 0.000,B 0.000,C 90.000,E1 135.729} C_DIS
LIN {X -0.053,Y -185.988,Z 870.735,A 0.000,B 0.000,C 90.000,E1 132.366} C_DIS
LIN {X 0.003,Y -190.620,Z 870.721,A 0.000,B 0.000,C 90.000,E1 129.850} C_DIS
LIN {X 0.024,Y -193.145,Z 870.713,A 0.000,B 0.000,C 90.000,E1 128.338} C_DIS
LIN {X 0.001,Y -294.441,Z 870.713,A 0.000,B 0.000,C 90.000,E1 128.338} C_DIS
LIN {X 0.113,Y -298.880,Z 870.712,A 0.000,B 0.000,C 90.000,E1 128.177} C_DIS
LIN {X 0.008,Y -302.072,Z 870.711,A 0.000,B 0.000,C 90.000,E1 127.971} C_DIS
LIN {X 0.125,Y -305.758,Z 870.709,A 0.000,B 0.000,C 90.000,E1 127.523} C_DIS
LIN {X -0.026,Y -307.664,Z 870.707,A 0.000,B 0.000,C 90.000,E1 127.237} C_DIS
LIN {X 0.006,Y -309.155,Z 870.705,A 0.000,B 0.000,C 90.000,E1 126.916} C_DIS
LIN {X 0.038,Y -310.376,Z 870.703,A 0.000,B 0.000,C 90.000,E1 126.583} C_DIS
LIN {X -0.010,Y -321.535,Z 870.684,A 0.000,B 0.000,C 90.000,E1 123.038} C_DIS
LIN {X -0.130,Y -332.022,Z 870.668,A 0.000,B 0.000,C 90.000,E1 120.207} C_DIS
LIN {X -0.004,Y -343.867,Z 870.652,A 0.000,B 0.000,C 90.000,E1 117.385} C_DIS
LIN {X -0.007,Y -357.171,Z 870.637,A 0.000,B 0.000,C 90.000,E1 114.643} C_DIS
LIN {X -0.023,Y -370.321,Z 870.624,A 0.000,B 0.000,C 90.000,E1 112.259} C_DIS
LIN {X -0.132,Y -384.812,Z 870.611,A 0.000,B 0.000,C 90.000,E1 109.939} C_DIS
LIN {X 0.001,Y -400.749,Z 870.598,A 0.000,B 0.000,C 90.000,E1 107.638} C_DIS
LIN {X -0.096,Y -418.246,Z 870.586,A 0.000,B 0.000,C 90.000,E1 105.426} C_DIS
LIN {X 0.044,Y -437.401,Z 870.574,A 0.000,B 0.000,C 90.000,E1 103.244} C_DIS
LIN {X -0.126,Y -457.537,Z 870.562,A 0.000,B 0.000,C 90.000,E1 101.243} C_DIS
LIN {X 0.206,Y -467.724,Z 870.557,A 0.000,B 0.000,C 90.000,E1 100.254} C_DIS
LIN {X 0.237,Y -469.654,Z 870.556,A 0.000,B 0.000,C 90.000,E1 100.018} C_DIS
LIN {X 0.007,Y -471.253,Z 870.554,A 0.000,B 0.000,C 90.000,E1 99.792} C_DIS
LIN {X -0.145,Y -472.452,Z 870.553,A 0.000,B 0.000,C 90.000,E1 99.557} C_DIS
LIN {X 0.036,Y -473.911,Z 870.550,A 0.000,B 0.000,C 90.000,E1 99.029} C_DIS
LIN {X 0.149,Y -474.337,Z 870.547,A 0.000,B 0.000,C 90.000,E1 98.511} C_DIS
LIN {X -0.197,Y -473.800,Z 870.545,A 0.000,B 0.000,C 90.000,E1 98.049} C_DIS
LIN {X -0.069,Y -472.220,Z 870.542,A 0.000,B 0.000,C 90.000,E1 97.530} C_DIS
LIN {X -0.209,Y -470.956,Z 870.540,A 0.000,B 0.000,C 90.000,E1 97.296} C_DIS
LIN {X -0.052,Y -453.443,Z 870.525,A 0.000,B 0.000,C 90.000,E1 94.473} C_DIS
LIN {X 0.082,Y -442.966,Z 870.515,A 0.000,B 0.000,C 90.000,E1 92.636} C_DIS
LIN {X -0.174,Y -433.550,Z 870.506,A 0.000,B 0.000,C 90.000,E1 91.088} C_DIS
LIN {X -0.164,Y -423.951,Z 870.497,A 0.000,B 0.000,C 90.000,E1 89.484} C_DIS
LIN {X 0.199,Y -412.511,Z 870.486,A 0.000,B 0.000,C 90.000,E1 87.535} C_DIS
LIN {X -0.073,Y -401.119,Z 870.476,A 0.000,B 0.000,C 90.000,E1 85.641} C_DIS
LIN {X -0.088,Y -388.209,Z 870.463,A 0.000,B 0.000,C 90.000,E1 83.394} C_DIS
LIN {X 0.001,Y -377.034,Z 870.452,A 0.000,B 0.000,C 90.000,E1 81.376} C_DIS
LIN {X -0.060,Y -364.388,Z 870.439,A 0.000,B 0.000,C 90.000,E1 79.050} C_DIS
LIN {X 0.124,Y -353.386,Z 870.428,A 0.000,B 0.000,C 90.000,E1 76.937} C_DIS
LIN {X 0.157,Y -342.400,Z 870.416,A 0.000,B 0.000,C 90.000,E1 74.810} C_DIS
LIN {X -0.015,Y -328.639,Z 870.400,A 0.000,B 0.000,C 90.000,E1 72.054} C_DIS
LIN {X 0.024,Y -316.742,Z 870.386,A 0.000,B 0.000,C 90.000,E1 69.518} C_DIS
LIN {X 0.095,Y -305.244,Z 870.372,A 0.000,B 0.000,C 90.000,E1 66.922} C_DIS
LIN {X 0.121,Y -293.876,Z 870.357,A 0.000,B 0.000,C 90.000,E1 64.280} C_DIS
LIN {X -0.106,Y -284.021,Z 870.344,A 0.000,B 0.000,C 90.000,E1 61.975} C_DIS
LIN {X 0.049,Y -272.890,Z 870.329,A 0.000,B 0.000,C 90.000,E1 59.203} C_DIS
LIN {X -0.064,Y -259.603,Z 870.310,A 0.000,B 0.000,C 90.000,E1 55.722} C_DIS
LIN {X -0.006,Y -248.699,Z 870.292,A 0.000,B 0.000,C 90.000,E1 52.477} C_DIS
LIN {X 0.016,Y -238.895,Z 870.273,A 0.000,B 0.000,C 90.000,E1 49.175} C_DIS
LIN {X -0.003,Y -228.858,Z 870.252,A 0.000,B 0.000,C 90.000,E1 45.445} C_DIS
LIN {X 0.000,Y -219.514,Z 870.231,A 0.000,B 0.000,C 90.000,E1 41.634} C_DIS
LIN {X -0.047,Y -212.462,Z 870.214,A 0.000,B 0.000,C 90.000,E1 38.543} C_DIS
LIN {X -0.035,Y -205.916,Z 870.197,A 0.000,B 0.000,C 90.000,E1 35.391} C_DIS
LIN {X -0.085,Y -199.776,Z 870.179,A 0.000,B 0.000,C 90.000,E1 32.212} C_DIS
LIN {X 0.007,Y -194.216,Z 870.161,A 0.000,B 0.000,C 90.000,E1 28.949} C_DIS
LIN {X 0.023,Y -189.318,Z 870.143,A 0.000,B 0.000,C 90.000,E1 25.668} C_DIS
LIN {X -0.018,Y -184.174,Z 870.120,A 0.000,B 0.000,C 90.000,E1 21.535} C_DIS
LIN {X 0.025,Y -180.161,Z 870.096,A 0.000,B 0.000,C 90.000,E1 17.330} C_DIS
LIN {X 0.056,Y -176.826,Z 870.068,A 0.000,B 0.000,C 90.000,E1 12.243} C_DIS
LIN {X -0.003,Y -174.784,Z 870.025,A 0.000,B 0.000,C 90.000,E1 4.588} C_DIS
LIN {X 0.066,Y -176.507,Z 869.974,A 0.000,B 0.000,C 90.000,E1 355.241} C_DIS
LIN {X 0.030,Y -179.479,Z 869.945,A 0.000,B 0.000,C 90.000,E1 350.151} C_DIS
LIN {X 0.010,Y -183.140,Z 869.922,A 0.000,B 0.000,C 90.000,E1 345.936} C_DIS
LIN {X -0.033,Y -187.928,Z 869.899,A 0.000,B 0.000,C 90.000,E1 341.764} C_DIS
LIN {X -0.082,Y -192.525,Z 869.880,A 0.000,B 0.000,C 90.000,E1 338.465} C_DIS
LIN {X 0.052,Y -199.192,Z 869.857,A 0.000,B 0.000,C 90.000,E1 334.332} C_DIS
LIN {X -0.065,Y -206.531,Z 869.835,A 0.000,B 0.000,C 90.000,E1 330.333} C_DIS
LIN {X 0.025,Y -214.487,Z 869.813,A 0.000,B 0.000,C 90.000,E1 326.342} C_DIS
LIN {X 0.053,Y -221.508,Z 869.796,A 0.000,B 0.000,C 90.000,E1 323.210} C_DIS
LIN {X 0.075,Y -230.180,Z 869.776,A 0.000,B 0.000,C 90.000,E1 319.747} C_DIS
LIN {X -0.105,Y -237.598,Z 869.762,A 0.000,B 0.000,C 90.000,E1 317.148} C_DIS
LIN {X -0.155,Y -246.949,Z 869.745,A 0.000,B 0.000,C 90.000,E1 314.190} C_DIS
LIN {X 0.085,Y -258.478,Z 869.727,A 0.000,B 0.000,C 90.000,E1 310.862} C_DIS
LIN {X -0.005,Y -270.996,Z 869.709,A 0.000,B 0.000,C 90.000,E1 307.684} C_DIS
LIN {X -0.006,Y -284.723,Z 869.692,A 0.000,B 0.000,C 90.000,E1 304.565} C_DIS
LIN {X -0.105,Y -299.761,Z 869.675,A 0.000,B 0.000,C 90.000,E1 301.544} C_DIS
LIN {X 0.073,Y -312.472,Z 869.662,A 0.000,B 0.000,C 90.000,E1 299.205} C_DIS
LIN {X 0.149,Y -324.299,Z 869.652,A 0.000,B 0.000,C 90.000,E1 297.257} C_DIS
LIN {X -0.037,Y -346.264,Z 869.634,A 0.000,B 0.000,C 90.000,E1 294.155} C_DIS
LIN {X 0.117,Y -367.800,Z 869.619,A 0.000,B 0.000,C 90.000,E1 291.408} C_DIS
LIN {X 0.108,Y -393.439,Z 869.603,A 0.000,B 0.000,C 90.000,E1 288.544} C_DIS
LIN {X -0.108,Y -406.425,Z 869.596,A 0.000,B 0.000,C 90.000,E1 287.221} C_DIS
LIN {X 0.068,Y -416.666,Z 869.590,A 0.000,B 0.000,C 90.000,E1 286.134} C_DIS
LIN {X 0.201,Y -429.162,Z 869.582,A 0.000,B 0.000,C 90.000,E1 284.773} C_DIS
LIN {X -0.047,Y -441.171,Z 869.575,A 0.000,B 0.000,C 90.000,E1 283.467} C_DIS
LIN {X -0.038,Y -450.335,Z 869.569,A 0.000,B 0.000,C 90.000,E1 282.411} C_DIS
LIN {X -0.010,Y -458.845,Z 869.563,A 0.000,B 0.000,C 90.000,E1 281.366} C_DIS
LIN {X 0.215,Y -466.773,Z 869.557,A 0.000,B 0.000,C 90.000,E1 280.310} C_DIS
LIN {X -0.017,Y -474.026,Z 869.552,A 0.000,B 0.000,C 90.000,E1 279.321} C_DIS
LIN {X -0.043,Y -478.998,Z 869.548,A 0.000,B 0.000,C 90.000,E1 278.568} C_DIS
LIN {X -0.021,Y -483.221,Z 869.543,A 0.000,B 0.000,C 90.000,E1 277.814} C_DIS
LIN {X -0.028,Y -486.732,Z 869.539,A 0.000,B 0.000,C 90.000,E1 277.068} C_DIS
LIN {X 0.172,Y -488.665,Z 869.536,A 0.000,B 0.000,C 90.000,E1 276.549} C_DIS
LIN {X -0.109,Y -490.299,Z 869.534,A 0.000,B 0.000,C 90.000,E1 276.087} C_DIS
LIN {X 0.109,Y -491.549,Z 869.531,A 0.000,B 0.000,C 90.000,E1 275.568} C_DIS
LIN {X -0.155,Y -492.465,Z 869.528,A 0.000,B 0.000,C 90.000,E1 275.106} C_DIS
LIN {X 0.075,Y -492.985,Z 869.526,A 0.000,B 0.000,C 90.000,E1 274.588} C_DIS
LIN {X -0.218,Y -493.122,Z 869.523,A 0.000,B 0.000,C 90.000,E1 274.131} C_DIS
LIN {X 0.021,Y -492.820,Z 869.520,A 0.000,B 0.000,C 90.000,E1 273.612} C_DIS
LIN {X 0.256,Y -492.043,Z 869.517,A 0.000,B 0.000,C 90.000,E1 273.094} C_DIS
LIN {X -0.030,Y -490.825,Z 869.515,A 0.000,B 0.000,C 90.000,E1 272.636} C_DIS
LIN {X 0.175,Y -489.100,Z 869.512,A 0.000,B 0.000,C 90.000,E1 272.121} C_DIS
LIN {X -0.099,Y -486.865,Z 869.509,A 0.000,B 0.000,C 90.000,E1 271.661} C_DIS
LIN {X 0.082,Y -484.072,Z 869.506,A 0.000,B 0.000,C 90.000,E1 271.146} C_DIS
LIN {X -0.234,Y -480.541,Z 869.504,A 0.000,B 0.000,C 90.000,E1 270.688} C_DIS
LIN {X -0.084,Y -476.239,Z 869.501,A 0.000,B 0.000,C 90.000,E1 270.172} C_DIS
LIN {X 0.042,Y -471.032,Z 869.498,A 0.000,B 0.000,C 90.000,E1 269.656} C_DIS
LIN {X -0.023,Y -465.268,Z 869.496,A 0.000,B 0.000,C 90.000,E1 269.198} C_DIS
LIN {X -0.151,Y -458.899,Z 869.493,A 0.000,B 0.000,C 90.000,E1 268.797} C_DIS
LIN {X 0.199,Y -452.020,Z 869.491,A 0.000,B 0.000,C 90.000,E1 268.396} C_DIS
LIN {X 0.171,Y -444.660,Z 869.490,A 0.000,B 0.000,C 90.000,E1 268.108} C_DIS
LIN {X 0.193,Y -437.404,Z 869.488,A 0.000,B 0.000,C 90.000,E1 267.879} C_DIS
LIN {X 0.132,Y -429.487,Z 869.487,A 0.000,B 0.000,C 90.000,E1 267.707} C_DIS
LIN {X -0.041,Y -419.563,Z 869.487,A 0.000,B 0.000,C 90.000,E1 267.593} C_DIS
LIN {X 0.061,Y -412.551,Z 869.486,A 0.000,B 0.000,C 90.000,E1 267.535} C_DIS
LIN {X -0.007,Y -181.055,Z 869.486,A 0.000,B 0.000,C 90.000,E1 267.535} C_DIS
LIN {X 0.068,Y -180.856,Z 869.472,A 0.000,B 0.000,C 90.000,E1 264.951} C_DIS
LIN {X -0.058,Y -178.967,Z 869.444,A 0.000,B 0.000,C 90.000,E1 259.926} C_DIS
LIN {X -0.047,Y -177.920,Z 869.435,A 0.000,B 0.000,C 90.000,E1 258.229} C_DIS
LIN {X -0.032,Y -175.556,Z 869.411,A 0.000,B 0.000,C 90.000,E1 253.976} C_DIS
LIN {X -0.025,Y -172.287,Z 869.387,A 0.000,B 0.000,C 90.000,E1 249.699} C_DIS
LIN {X -0.047,Y -171.765,Z 869.382,A 0.000,B 0.000,C 90.000,E1 248.847} C_DIS
LIN {X 0.032,Y -167.366,Z 869.354,A 0.000,B 0.000,C 90.000,E1 243.640} C_DIS
LIN {X -0.035,Y -166.757,Z 869.349,A 0.000,B 0.000,C 90.000,E1 242.794} C_DIS
LIN {X 0.024,Y -162.735,Z 869.325,A 0.000,B 0.000,C 90.000,E1 238.408} C_DIS
LIN {X 0.085,Y -161.426,Z 869.315,A 0.000,B 0.000,C 90.000,E1 236.628} C_DIS
LIN {X -0.094,Y -157.419,Z 869.290,A 0.000,B 0.000,C 90.000,E1 232.271} C_DIS
LIN {X 0.059,Y -155.422,Z 869.275,A 0.000,B 0.000,C 90.000,E1 229.542} C_DIS
LIN {X -0.010,Y -151.747,Z 869.250,A 0.000,B 0.000,C 90.000,E1 225.081} C_DIS
LIN {X 0.001,Y -149.947,Z 869.235,A 0.000,B 0.000,C 90.000,E1 222.366} C_DIS
LIN {X 0.029,Y -146.791,Z 869.210,A 0.000,B 0.000,C 90.000,E1 217.810} C_DIS
LIN {X -0.070,Y -145.365,Z 869.195,A 0.000,B 0.000,C 90.000,E1 215.105} C_DIS
LIN {X 0.046,Y -142.432,Z 869.164,A 0.000,B 0.000,C 90.000,E1 209.539} C_DIS
LIN {X -0.031,Y -141.421,Z 869.149,A 0.000,B 0.000,C 90.000,E1 206.796} C_DIS
LIN {X -0.049,Y -139.362,Z 869.113,A 0.000,B 0.000,C 90.000,E1 200.301} C_DIS
LIN {X 0.070,Y -138.806,Z 869.097,A 0.000,B 0.000,C 90.000,E1 197.457} C_DIS
LIN {X -0.012,Y -138.350,Z 869.056,A 0.000,B 0.000,C 90.000,E1 190.018} C_DIS
LIN {X -0.036,Y -139.544,Z 869.004,A 0.000,B 0.000,C 90.000,E1 180.688} C_DIS
LIN {X 0.057,Y -141.245,Z 868.973,A 0.000,B 0.000,C 90.000,E1 175.065} C_DIS
LIN {X 0.015,Y -142.614,Z 868.957,A 0.000,B 0.000,C 90.000,E1 172.299} C_DIS
LIN {X -0.032,Y -144.930,Z 868.932,A 0.000,B 0.000,C 90.000,E1 167.701} C_DIS
LIN {X -0.040,Y -147.559,Z 868.911,A 0.000,B 0.000,C 90.000,E1 164.031} C_DIS
LIN {X -0.009,Y -150.165,Z 868.891,A 0.000,B 0.000,C 90.000,E1 160.369} C_DIS
LIN {X 0.000,Y -153.538,Z 868.871,A 0.000,B 0.000,C 90.000,E1 156.741} C_DIS
LIN {X 0.053,Y -156.955,Z 868.851,A 0.000,B 0.000,C 90.000,E1 153.127} C_DIS
LIN {X -0.012,Y -161.062,Z 868.831,A 0.000,B 0.000,C 90.000,E1 149.587} C_DIS
LIN {X 0.073,Y -163.170,Z 868.821,A 0.000,B 0.000,C 90.000,E1 147.788} C_DIS
LIN {X -0.056,Y -167.590,Z 868.802,A 0.000,B 0.000,C 90.000,E1 144.322} C_DIS
LIN {X -0.011,Y -171.419,Z 868.787,A 0.000,B 0.000,C 90.000,E1 141.698} C_DIS
LIN {X 0.028,Y -176.337,Z 868.768,A 0.000,B 0.000,C 90.000,E1 138.243} C_DIS
LIN {X -0.104,Y -180.625,Z 868.754,A 0.000,B 0.000,C 90.000,E1 135.729} C_DIS
LIN {X 0.010,Y -186.027,Z 868.735,A 0.000,B 0.000,C 90.000,E1 132.324} C_DIS
LIN {X 0.073,Y -190.662,Z 868.721,A 0.000,B 0.000,C 90.000,E1 129.806} C_DIS
LIN {X -0.084,Y -193.122,Z 868.713,A 0.000,B 0.000,C 90.000,E1 128.382} C_DIS
LIN {X 0.068,Y -293.975,Z 868.713,A 0.000,B 0.000,C 90.000,E1 128.338} C_DIS
LIN {X -0.036,Y -295.518,Z 868.713,A 0.000,B 0.000,C 90.000,E1 128.338} C_DIS
LIN {X -0.005,Y -299.407,Z 868.712,A 0.000,B 0.000,C 90.000,E1 128.177} C_DIS
LIN {X -0.047,Y -302.616,Z 868.711,A 0.000,B 0.000,C 90.000,E1 127.935} C_DIS
LIN {X 0.127,Y -306.305,Z 868.708,A 0.000,B 0.000,C 90.000,E1 127.443} C_DIS
LIN {X -0.103,Y -308.148,Z 868.706,A 0.000,B 0.000,C 90.000,E1 127.156} C_DIS
LIN {X 0.099,Y -309.584,Z 868.704,A 0.000,B 0.000,C 90.000,E1 126.790} C_DIS
LIN {X -0.080,Y -311.649,Z 868.701,A 0.000,B 0.000,C 90.000,E1 126.171} C_DIS
LIN {X -0.163,Y -321.879,Z 868.683,A 0.000,B 0.000,C 90.000,E1 122.959} C_DIS
LIN {X 0.004,Y -332.413,Z 868.667,A 0.000,B 0.000,C 90.000,E1 120.079} C_DIS
LIN {X 0.148,Y -344.312,Z 868.652,A 0.000,B 0.000,C 90.000,E1 117.257} C_DIS
LIN {X 0.163,Y -357.672,Z 868.636,A 0.000,B 0.000,C 90.000,E1 114.515} C_DIS
LIN {X 0.024,Y -370.875,Z 868.623,A 0.000,B 0.000,C 90.000,E1 112.153} C_DIS
LIN {X 0.075,Y -385.424,Z 868.610,A 0.000,B 0.000,C 90.000,E1 109.812} C_DIS
LIN {X 0.105,Y -401.424,Z 868.597,A 0.000,B 0.000,C 90.000,E1 107.528} C_DIS
LIN {X 0.039,Y -418.988,Z 868.585,A 0.000,B 0.000,C 90.000,E1 105.315} C_DIS
LIN {X -0.110,Y -438.210,Z 868.573,A 0.000,B 0.000,C 90.000,E1 103.175} C_DIS
LIN {X 0.120,Y -458.370,Z 868.562,A 0.000,B 0.000,C 90.000,E1 101.130} C_DIS
LIN {X -0.011,Y -466.087,Z 868.558,A 0.000,B 0.000,C 90.000,E1 100.433} C_DIS
LIN {X 0.027,Y -468.414,Z 868.557,A 0.000,B 0.000,C 90.000,E1 100.197} C_DIS
LIN {X 0.065,Y -470.174,Z 868.555,A 0.000,B 0.000,C 90.000,E1 99.962} C_DIS
LIN {X -0.085,Y -471.643,Z 868.554,A 0.000,B 0.000,C 90.000,E1 99.726} C_DIS
LIN {X 0.153,Y -472.739,Z 868.553,A 0.000,B 0.000,C 90.000,E1 99.443} C_DIS
LIN {X -0.131,Y -474.035,Z 868.550,A 0.000,B 0.000,C 90.000,E1 98.973} C_DIS
LIN {X -0.016,Y -474.320,Z 868.547,A 0.000,B 0.000,C 90.000,E1 98.454} C_DIS
LIN {X 0.110,Y -473.641,Z 868.544,A 0.000,B 0.000,C 90.000,E1 97.936} C_DIS
LIN {X -0.169,Y -471.891,Z 868.541,A 0.000,B 0.000,C 90.000,E1 97.466} C_DIS
LIN {X 0.096,Y -470.516,Z 868.540,A 0.000,B 0.000,C 90.000,E1 97.182} C_DIS
LIN {X 0.012,Y -454.526,Z 868.526,A 0.000,B 0.000,C 90.000,E1 94.645} C_DIS
LIN {X 0.168,Y -444.048,Z 868.516,A 0.000,B 0.000,C 90.000,E1 92.808} C_DIS
LIN {X -0.073,Y -434.705,Z 868.507,A 0.000,B 0.000,C 90.000,E1 91.260} C_DIS
LIN {X -0.045,Y -425.098,Z 868.498,A 0.000,B 0.000,C 90.000,E1 89.656} C_DIS
LIN {X -0.079,Y -413.683,Z 868.488,A 0.000,B 0.000,C 90.000,E1 87.764} C_DIS
LIN {X 0.139,Y -400.646,Z 868.475,A 0.000,B 0.000,C 90.000,E1 85.527} C_DIS
LIN {X 0.102,Y -387.731,Z 868.463,A 0.000,B 0.000,C 90.000,E1 83.280} C_DIS
LIN {X -0.188,Y -374.960,Z 868.450,A 0.000,B 0.000,C 90.000,E1 81.027} C_DIS
LIN {X 0.136,Y -362.365,Z 868.437,A 0.000,B 0.000,C 90.000,E1 78.634} C_DIS
LIN {X -0.140,Y -351.384,Z 868.425,A 0.000,B 0.000,C 90.000,E1 76.589} C_DIS
LIN {X -0.153,Y -338.921,Z 868.412,A 0.000,B 0.000,C 90.000,E1 74.157} C_DIS
LIN {X 0.043,Y -326.750,Z 868.398,A 0.000,B 0.000,C 90.000,E1 71.638} C_DIS
LIN {X 0.139,Y -314.940,Z 868.384,A 0.000,B 0.000,C 90.000,E1 69.082} C_DIS
LIN {X -0.020,Y -304.922,Z 868.371,A 0.000,B 0.000,C 90.000,E1 66.847} C_DIS
LIN {X 0.008,Y -293.598,Z 868.357,A 0.000,B 0.000,C 90.000,E1 64.204} C_DIS
LIN {X 0.036,Y -283.792,Z 868.344,A 0.000,B 0.000,C 90.000,E1 61.847} C_DIS
LIN {X -0.056,Y -272.727,Z 868.328,A 0.000,B 0.000,C 90.000,E1 59.125} C_DIS
LIN {X 0.051,Y -259.524,Z 868.309,A 0.000,B 0.000,C 90.000,E1 55.595} C_DIS
LIN {X 0.098,Y -248.703,Z 868.291,A 0.000,B 0.000,C 90.000,E1 52.351} C_DIS
LIN {X -0.071,Y -238.943,Z 868.273,A 0.000,B 0.000,C 90.000,E1 49.094} C_DIS
LIN {X 0.077,Y -228.916,Z 868.252,A 0.000,B 0.000,C 90.000,E1 45.324} C_DIS
LIN {X 0.068,Y -219.593,Z 868.231,A 0.000,B 0.000,C 90.000,E1 41.515} C_DIS
LIN {X -0.006,Y -210.864,Z 868.209,A 0.000,B 0.000,C 90.000,E1 37.649} C_DIS
LIN {X -0.055,Y -202.904,Z 868.187,A 0.000,B 0.000,C 90.000,E1 33.706} C_DIS
LIN {X 0.045,Y -197.045,Z 868.169,A 0.000,B 0.000,C 90.000,E1 30.463} C_DIS
LIN {X 0.047,Y -191.827,Z 868.151,A 0.000,B 0.000,C 90.000,E1 27.206} C_DIS
LIN {X -0.081,Y -187.292,Z 868.133,A 0.000,B 0.000,C 90.000,E1 23.951} C_DIS
LIN {X 0.017,Y -182.617,Z 868.110,A 0.000,B 0.000,C 90.000,E1 19.758} C_DIS
LIN {X 0.019,Y -179.081,Z 868.086,A 0.000,B 0.000,C 90.000,E1 15.552} C_DIS
LIN {X -0.061,Y -176.340,Z 868.058,A 0.000,B 0.000,C 90.000,E1 10.489} C_DIS
LIN {X -0.054,Y -177.262,Z 867.969,A 0.000,B 0.000,C 90.000,E1 354.432} C_DIS
LIN {X 0.054,Y -179.848,Z 867.945,A 0.000,B 0.000,C 90.000,E1 350.151} C_DIS
LIN {X 0.045,Y -183.514,Z 867.922,A 0.000,B 0.000,C 90.000,E1 345.936} C_DIS
LIN {X 0.016,Y -188.304,Z 867.899,A 0.000,B 0.000,C 90.000,E1 341.764} C_DIS
LIN {X -0.022,Y -192.874,Z 867.880,A 0.000,B 0.000,C 90.000,E1 338.465} C_DIS
LIN {X 0.038,Y -199.524,Z 867.858,A 0.000,B 0.000,C 90.000,E1 334.357} C_DIS
LIN {X 0.021,Y -206.838,Z 867.835,A 0.000,B 0.000,C 90.000,E1 330.333} C_DIS
LIN {X 0.005,Y -214.769,Z 867.813,A 0.000,B 0.000,C 90.000,E1 326.373} C_DIS
LIN {X -0.015,Y -221.767,Z 867.796,A 0.000,B 0.000,C 90.000,E1 323.256} C_DIS
LIN {X 0.048,Y -230.438,Z 867.777,A 0.000,B 0.000,C 90.000,E1 319.784} C_DIS
LIN {X -0.007,Y -238.964,Z 867.760,A 0.000,B 0.000,C 90.000,E1 316.782} C_DIS
LIN {X 0.153,Y -248.393,Z 867.743,A 0.000,B 0.000,C 90.000,E1 313.785} C_DIS
LIN {X 0.077,Y -259.986,Z 867.725,A 0.000,B 0.000,C 90.000,E1 310.539} C_DIS
LIN {X 0.027,Y -272.593,Z 867.708,A 0.000,B 0.000,C 90.000,E1 307.363} C_DIS
LIN {X 0.055,Y -286.362,Z 867.690,A 0.000,B 0.000,C 90.000,E1 304.246} C_DIS
LIN {X 0.095,Y -301.498,Z 867.673,A 0.000,B 0.000,C 90.000,E1 301.209} C_DIS
LIN {X -0.113,Y -314.315,Z 867.661,A 0.000,B 0.000,C 90.000,E1 298.949} C_DIS
LIN {X -0.006,Y -326.245,Z 867.650,A 0.000,B 0.000,C 90.000,E1 297.001} C_DIS
LIN {X -0.143,Y -345.996,Z 867.634,A 0.000,B 0.000,C 90.000,E1 294.207} C_DIS
LIN {X 0.068,Y -369.882,Z 867.618,A 0.000,B 0.000,C 90.000,E1 291.153} C_DIS
LIN {X 0.012,Y -395.658,Z 867.602,A 0.000,B 0.000,C 90.000,E1 288.308} C_DIS
LIN {X 0.070,Y -411.259,Z 867.593,A 0.000,B 0.000,C 90.000,E1 286.677} C_DIS
LIN {X 0.127,Y -421.372,Z 867.587,A 0.000,B 0.000,C 90.000,E1 285.607} C_DIS
LIN {X 0.101,Y -431.278,Z 867.581,A 0.000,B 0.000,C 90.000,E1 284.537} C_DIS
LIN {X -0.127,Y -443.235,Z 867.573,A 0.000,B 0.000,C 90.000,E1 283.231} C_DIS
LIN {X -0.095,Y -452.238,Z 867.568,A 0.000,B 0.000,C 90.000,E1 282.175} C_DIS
LIN {X -0.046,Y -460.660,Z 867.562,A 0.000,B 0.000,C 90.000,E1 281.130} C_DIS
LIN {X 0.198,Y -468.407,Z 867.556,A 0.000,B 0.000,C 90.000,E1 280.074} C_DIS
LIN {X -0.094,Y -475.570,Z 867.550,A 0.000,B 0.000,C 90.000,E1 279.095} C_DIS
LIN {X -0.098,Y -480.291,Z 867.546,A 0.000,B 0.000,C 90.000,E1 278.341} C_DIS
LIN {X -0.066,Y -484.336,Z 867.542,A 0.000,B 0.000,C 90.000,E1 277.587} C_DIS
LIN {X 0.116,Y -486.629,Z 867.539,A 0.000,B 0.000,C 90.000,E1 277.068} C_DIS
LIN {X -0.170,Y -488.557,Z 867.537,A 0.000,B 0.000,C 90.000,E1 276.606} C_DIS
LIN {X 0.036,Y -490.193,Z 867.534,A 0.000,B 0.000,C 90.000,E1 276.087} C_DIS
LIN {X -0.237,Y -491.499,Z 867.531,A 0.000,B 0.000,C 90.000,E1 275.625} C_DIS
LIN {X -0.012,Y -492.419,Z 867.528,A 0.000,B 0.000,C 90.000,E1 275.106} C_DIS
LIN {X 0.219,Y -492.974,Z 867.526,A 0.000,B 0.000,C 90.000,E1 274.588} C_DIS
LIN {X -0.074,Y -493.131,Z 867.523,A 0.000,B 0.000,C 90.000,E1 274.131} C_DIS
LIN {X 0.164,Y -492.833,Z 867.520,A 0.000,B 0.000,C 90.000,E1 273.612} C_DIS
LIN {X -0.119,Y -492.121,Z 867.517,A 0.000,B 0.000,C 90.000,E1 273.154} C_DIS
LIN {X 0.113,Y -490.934,Z 867.515,A 0.000,B 0.000,C 90.000,E1 272.636} C_DIS
LIN {X -0.172,Y -489.247,Z 867.512,A 0.000,B 0.000,C 90.000,E1 272.178} C_DIS
LIN {X 0.043,Y -487.066,Z 867.509,A 0.000,B 0.000,C 90.000,E1 271.661} C_DIS
LIN {X 0.224,Y -484.295,Z 867.507,A 0.000,B 0.000,C 90.000,E1 271.146} C_DIS
LIN {X -0.091,Y -480.841,Z 867.504,A 0.000,B 0.000,C 90.000,E1 270.688} C_DIS
LIN {X 0.060,Y -476.621,Z 867.501,A 0.000,B 0.000,C 90.000,E1 270.172} C_DIS
LIN {X -0.114,Y -474.237,Z 867.500,A 0.000,B 0.000,C 90.000,E1 269.943} C_DIS
LIN {X 0.126,Y -468.825,Z 867.497,A 0.000,B 0.000,C 90.000,E1 269.427} C_DIS
LIN {X 0.213,Y -462.822,Z 867.494,A 0.000,B 0.000,C 90.000,E1 268.969} C_DIS
LIN {X -0.177,Y -456.311,Z 867.492,A 0.000,B 0.000,C 90.000,E1 268.625} C_DIS
LIN {X -0.061,Y -449.258,Z 867.490,A 0.000,B 0.000,C 90.000,E1 268.282} C_DIS
LIN {X 0.119,Y -441.900,Z 867.489,A 0.000,B 0.000,C 90.000,E1 267.993} C_DIS
LIN {X -0.161,Y -434.132,Z 867.488,A 0.000,B 0.000,C 90.000,E1 267.822} C_DIS
LIN {X -0.061,Y -425.778,Z 867.487,A 0.000,B 0.000,C 90.000,E1 267.650} C_DIS
LIN {X -0.138,Y -420.607,Z 867.487,A 0.000,B 0.000,C 90.000,E1 267.593} C_DIS
LIN {X -0.133,Y -409.979,Z 867.486,A 0.000,B 0.000,C 90.000,E1 267.535} C_DIS
LIN {X 0.086,Y -181.052,Z 867.486,A 0.000,B 0.000,C 90.000,E1 267.478} C_DIS
LIN {X 0.011,Y -180.851,Z 867.472,A 0.000,B 0.000,C 90.000,E1 264.951} C_DIS
LIN {X 0.093,Y -178.961,Z 867.444,A 0.000,B 0.000,C 90.000,E1 259.859} C_DIS
LIN {X -0.015,Y -177.368,Z 867.430,A 0.000,B 0.000,C 90.000,E1 257.353} C_DIS
LIN {X 0.080,Y -175.542,Z 867.411,A 0.000,B 0.000,C 90.000,E1 253.921} C_DIS
LIN {X -0.080,Y -172.275,Z 867.387,A 0.000,B 0.000,C 90.000,E1 249.699} C_DIS
LIN {X -0.041,Y -171.754,Z 867.382,A 0.000,B 0.000,C 90.000,E1 248.827} C_DIS
LIN {X -0.023,Y -167.353,Z 867.354,A 0.000,B 0.000,C 90.000,E1 243.640} C_DIS
LIN {X 0.059,Y -166.741,Z 867.349,A 0.000,B 0.000,C 90.000,E1 242.743} C_DIS
LIN {X -0.029,Y -162.721,Z 867.324,A 0.000,B 0.000,C 90.000,E1 238.408} C_DIS
LIN {X 0.033,Y -161.411,Z 867.315,A 0.000,B 0.000,C 90.000,E1 236.628} C_DIS
LIN {X 0.074,Y -157.405,Z 867.290,A 0.000,B 0.000,C 90.000,E1 232.190} C_DIS
LIN {X 0.007,Y -155.404,Z 867.275,A 0.000,B 0.000,C 90.000,E1 229.542} C_DIS
LIN {X -0.062,Y -151.734,Z 867.250,A 0.000,B 0.000,C 90.000,E1 225.081} C_DIS
LIN {X -0.050,Y -149.930,Z 867.235,A 0.000,B 0.000,C 90.000,E1 222.366} C_DIS
LIN {X -0.022,Y -146.780,Z 867.210,A 0.000,B 0.000,C 90.000,E1 217.810} C_DIS
LIN {X 0.082,Y -145.352,Z 867.195,A 0.000,B 0.000,C 90.000,E1 215.025} C_DIS
LIN {X -0.003,Y -142.424,Z 867.164,A 0.000,B 0.000,C 90.000,E1 209.539} C_DIS
LIN {X 0.046,Y -141.412,Z 867.149,A 0.000,B 0.000,C 90.000,E1 206.744} C_DIS
LIN {X 0.033,Y -139.359,Z 867.113,A 0.000,B 0.000,C 90.000,E1 200.248} C_DIS
LIN {X 0.021,Y -138.801,Z 867.097,A 0.000,B 0.000,C 90.000,E1 197.457} C_DIS
LIN {X -0.061,Y -138.349,Z 867.056,A 0.000,B 0.000,C 90.000,E1 190.018} C_DIS
LIN {X -0.046,Y -139.367,Z 867.009,A 0.000,B 0.000,C 90.000,E1 181.604} C_DIS
LIN {X 0.007,Y -141.254,Z 866.973,A 0.000,B 0.000,C 90.000,E1 175.065} C_DIS
LIN {X -0.034,Y -142.622,Z 866.957,A 0.000,B 0.000,C 90.000,E1 172.299} C_DIS
LIN {X 0.059,Y -144.942,Z 866.932,A 0.000,B 0.000,C 90.000,E1 167.645} C_DIS
LIN {X 0.051,Y -147.571,Z 866.911,A 0.000,B 0.000,C 90.000,E1 163.976} C_DIS
LIN {X -0.059,Y -150.181,Z 866.891,A 0.000,B 0.000,C 90.000,E1 160.369} C_DIS
LIN {X -0.052,Y -153.558,Z 866.871,A 0.000,B 0.000,C 90.000,E1 156.741} C_DIS
LIN {X 0.000,Y -156.975,Z 866.851,A 0.000,B 0.000,C 90.000,E1 153.127} C_DIS
LIN {X 0.074,Y -161.086,Z 866.831,A 0.000,B 0.000,C 90.000,E1 149.537} C_DIS
LIN {X 0.020,Y -163.192,Z 866.821,A 0.000,B 0.000,C 90.000,E1 147.788} C_DIS
LIN {X 0.025,Y -167.616,Z 866.802,A 0.000,B 0.000,C 90.000,E1 144.276} C_DIS
LIN {X -0.066,Y -171.442,Z 866.787,A 0.000,B 0.000,C 90.000,E1 141.698} C_DIS
LIN {X -0.029,Y -176.364,Z 866.768,A 0.000,B 0.000,C 90.000,E1 138.243} C_DIS
LIN {X 0.094,Y -180.656,Z 866.754,A 0.000,B 0.000,C 90.000,E1 135.648} C_DIS
LIN {X 0.077,Y -186.058,Z 866.735,A 0.000,B 0.000,C 90.000,E1 132.285} C_DIS
LIN {X 0.014,Y -190.695,Z 866.721,A 0.000,B 0.000,C 90.000,E1 129.806} C_DIS
LIN {X -0.048,Y -193.103,Z 866.713,A 0.000,B 0.000,C 90.000,E1 128.382} C_DIS
LIN {X -0.107,Y -293.717,Z 866.713,A 0.000,B 0.000,C 90.000,E1 128.382} C_DIS
LIN {X 0.018,Y -295.418,Z 866.713,A 0.000,B 0.000,C 90.000,E1 128.338} C_DIS
LIN {X -0.097,Y -299.800,Z 866.712,A 0.000,B 0.000,C 90.000,E1 128.177} C_DIS
LIN {X 0.036,Y -302.962,Z 866.711,A 0.000,B 0.000,C 90.000,E1 127.890} C_DIS
LIN {X -0.164,Y -306.654,Z 866.708,A 0.000,B 0.000,C 90.000,E1 127.443} C_DIS
LIN {X 0.037,Y -308.406,Z 866.706,A 0.000,B 0.000,C 90.000,E1 127.076} C_DIS
LIN {X 0.055,Y -309.777,Z 866.704,A 0.000,B 0.000,C 90.000,E1 126.744} C_DIS
LIN {X -0.099,Y -320.951,Z 866.684,A 0.000,B 0.000,C 90.000,E1 123.214} C_DIS
LIN {X 0.031,Y -331.366,Z 866.669,A 0.000,B 0.000,C 90.000,E1 120.335} C_DIS
LIN {X 0.146,Y -343.132,Z 866.653,A 0.000,B 0.000,C 90.000,E1 117.513} C_DIS
LIN {X 0.122,Y -356.355,Z 866.638,A 0.000,B 0.000,C 90.000,E1 114.771} C_DIS
LIN {X 0.093,Y -369.424,Z 866.624,A 0.000,B 0.000,C 90.000,E1 112.386} C_DIS
LIN {X -0.031,Y -383.829,Z 866.611,A 0.000,B 0.000,C 90.000,E1 110.066} C_DIS
LIN {X 0.086,Y -399.674,Z 866.599,A 0.000,B 0.000,C 90.000,E1 107.764} C_DIS
LIN {X -0.029,Y -417.071,Z 866.586,A 0.000,B 0.000,C 90.000,E1 105.552} C_DIS
LIN {X 0.171,Y -436.143,Z 866.574,A 0.000,B 0.000,C 90.000,E1 103.355} C_DIS
LIN {X -0.175,Y -456.244,Z 866.563,A 0.000,B 0.000,C 90.000,E1 101.366} C_DIS
LIN {X 0.203,Y -466.504,Z 866.558,A 0.000,B 0.000,C 90.000,E1 100.366} C_DIS
LIN {X 0.162,Y -468.733,Z 866.556,A 0.000,B 0.000,C 90.000,E1 100.141} C_DIS
LIN {X 0.203,Y -470.418,Z 866.555,A 0.000,B 0.000,C 90.000,E1 99.905} C_DIS
LIN {X 0.055,Y -471.828,Z 866.554,A 0.000,B 0.000,C 90.000,E1 99.670} C_DIS
LIN {X -0.095,Y -472.876,Z 866.552,A 0.000,B 0.000,C 90.000,E1 99.434} C_DIS
LIN {X 0.012,Y -474.097,Z 866.550,A 0.000,B 0.000,C 90.000,E1 98.916} C_DIS
LIN {X 0.129,Y -474.312,Z 866.547,A 0.000,B 0.000,C 90.000,E1 98.398} C_DIS
LIN {X -0.214,Y -473.562,Z 866.544,A 0.000,B 0.000,C 90.000,E1 97.936} C_DIS
LIN {X -0.024,Y -471.728,Z 866.541,A 0.000,B 0.000,C 90.000,E1 97.409} C_DIS
LIN {X -0.226,Y -470.296,Z 866.540,A 0.000,B 0.000,C 90.000,E1 97.182} C_DIS
LIN {X 0.149,Y -454.314,Z 866.526,A 0.000,B 0.000,C 90.000,E1 94.588} C_DIS
LIN {X -0.144,Y -443.828,Z 866.516,A 0.000,B 0.000,C 90.000,E1 92.808} C_DIS
LIN {X 0.052,Y -434.493,Z 866.507,A 0.000,B 0.000,C 90.000,E1 91.203} C_DIS
LIN {X 0.073,Y -424.870,Z 866.498,A 0.000,B 0.000,C 90.000,E1 89.599} C_DIS
LIN {X 0.032,Y -413.467,Z 866.487,A 0.000,B 0.000,C 90.000,E1 87.707} C_DIS
LIN {X 0.191,Y -402.051,Z 866.477,A 0.000,B 0.000,C 90.000,E1 85.755} C_DIS
LIN {X 0.147,Y -389.096,Z 866.464,A 0.000,B 0.000,C 90.000,E1 83.514} C_DIS
LIN {X -0.063,Y -376.327,Z 866.451,A 0.000,B 0.000,C 90.000,E1 81.254} C_DIS
LIN {X -0.151,Y -362.162,Z 866.437,A 0.000,B 0.000,C 90.000,E1 78.634} C_DIS
LIN {X 0.001,Y -351.202,Z 866.425,A 0.000,B 0.000,C 90.000,E1 76.520} C_DIS
LIN {X -0.103,Y -338.768,Z 866.412,A 0.000,B 0.000,C 90.000,E1 74.102} C_DIS
LIN {X 0.082,Y -326.591,Z 866.398,A 0.000,B 0.000,C 90.000,E1 71.583} C_DIS
LIN {X -0.126,Y -314.817,Z 866.384,A 0.000,B 0.000,C 90.000,E1 69.082} C_DIS
LIN {X 0.002,Y -304.821,Z 866.371,A 0.000,B 0.000,C 90.000,E1 66.794} C_DIS
LIN {X 0.022,Y -293.536,Z 866.356,A 0.000,B 0.000,C 90.000,E1 64.152} C_DIS
LIN {X -0.074,Y -283.775,Z 866.343,A 0.000,B 0.000,C 90.000,E1 61.820} C_DIS
LIN {X -0.057,Y -272.766,Z 866.328,A 0.000,B 0.000,C 90.000,E1 59.076} C_DIS
LIN {X 0.043,Y -259.643,Z 866.309,A 0.000,B 0.000,C 90.000,E1 55.548} C_DIS
LIN {X 0.042,Y -248.883,Z 866.291,A 0.000,B 0.000,C 90.000,E1 52.316} C_DIS
LIN {X 0.072,Y -239.144,Z 866.272,A 0.000,B 0.000,C 90.000,E1 49.013} C_DIS
LIN {X -0.104,Y -229.123,Z 866.252,A 0.000,B 0.000,C 90.000,E1 45.324} C_DIS
LIN {X 0.067,Y -219.821,Z 866.230,A 0.000,B 0.000,C 90.000,E1 41.472} C_DIS
LIN {X 0.022,Y -212.784,Z 866.213,A 0.000,B 0.000,C 90.000,E1 38.382} C_DIS
LIN {X -0.019,Y -204.668,Z 866.191,A 0.000,B 0.000,C 90.000,E1 34.452} C_DIS
LIN {X -0.086,Y -197.281,Z 866.169,A 0.000,B 0.000,C 90.000,E1 30.463} C_DIS
LIN {X 0.013,Y -192.055,Z 866.151,A 0.000,B 0.000,C 90.000,E1 27.180} C_DIS
LIN {X -0.023,Y -187.510,Z 866.133,A 0.000,B 0.000,C 90.000,E1 23.898} C_DIS
LIN {X 0.034,Y -183.706,Z 866.114,A 0.000,B 0.000,C 90.000,E1 20.556} C_DIS
LIN {X -0.047,Y -179.958,Z 866.091,A 0.000,B 0.000,C 90.000,E1 16.386} C_DIS
LIN {X -0.019,Y -176.963,Z 866.063,A 0.000,B 0.000,C 90.000,E1 11.299} C_DIS
LIN {X -0.041,Y -177.620,Z 865.969,A 0.000,B 0.000,C 90.000,E1 354.432} C_DIS
LIN {X -0.034,Y -180.867,Z 865.941,A 0.000,B 0.000,C 90.000,E1 349.342} C_DIS
LIN {X 0.068,Y -184.772,Z 865.917,A 0.000,B 0.000,C 90.000,E1 345.102} C_DIS
LIN {X -0.042,Y -189.742,Z 865.894,A 0.000,B 0.000,C 90.000,E1 340.967} C_DIS
LIN {X -0.043,Y -194.501,Z 865.876,A 0.000,B 0.000,C 90.000,E1 337.667} C_DIS
LIN {X -0.034,Y -201.249,Z 865.853,A 0.000,B 0.000,C 90.000,E1 333.589} C_DIS
LIN {X 0.108,Y -207.129,Z 865.835,A 0.000,B 0.000,C 90.000,E1 330.333} C_DIS
LIN {X -0.074,Y -215.054,Z 865.813,A 0.000,B 0.000,C 90.000,E1 326.421} C_DIS
LIN {X -0.038,Y -222.027,Z 865.796,A 0.000,B 0.000,C 90.000,E1 323.290} C_DIS
LIN {X -0.007,Y -230.688,Z 865.777,A 0.000,B 0.000,C 90.000,E1 319.828} C_DIS
LIN {X -0.048,Y -239.189,Z 865.760,A 0.000,B 0.000,C 90.000,E1 316.824} C_DIS
LIN {X -0.056,Y -248.599,Z 865.744,A 0.000,B 0.000,C 90.000,E1 313.866} C_DIS
LIN {X -0.134,Y -260.145,Z 865.726,A 0.000,B 0.000,C 90.000,E1 310.620} C_DIS
LIN {X 0.028,Y -272.692,Z 865.708,A 0.000,B 0.000,C 90.000,E1 307.397} C_DIS
LIN {X 0.073,Y -286.419,Z 865.690,A 0.000,B 0.000,C 90.000,E1 304.278} C_DIS
LIN {X 0.026,Y -301.475,Z 865.674,A 0.000,B 0.000,C 90.000,E1 301.258} C_DIS
LIN {X 0.083,Y -314.223,Z 865.661,A 0.000,B 0.000,C 90.000,E1 298.949} C_DIS
LIN {X -0.094,Y -326.096,Z 865.650,A 0.000,B 0.000,C 90.000,E1 297.052} C_DIS
LIN {X 0.063,Y -343.466,Z 865.636,A 0.000,B 0.000,C 90.000,E1 294.515} C_DIS
LIN {X 0.067,Y -367.034,Z 865.619,A 0.000,B 0.000,C 90.000,E1 291.482} C_DIS
LIN {X -0.097,Y -395.116,Z 865.602,A 0.000,B 0.000,C 90.000,E1 288.362} C_DIS
LIN {X -0.039,Y -410.683,Z 865.593,A 0.000,B 0.000,C 90.000,E1 286.732} C_DIS
LIN {X 0.046,Y -420.800,Z 865.587,A 0.000,B 0.000,C 90.000,E1 285.662} C_DIS
LIN {X 0.025,Y -430.706,Z 865.581,A 0.000,B 0.000,C 90.000,E1 284.592} C_DIS
LIN {X 0.116,Y -442.709,Z 865.574,A 0.000,B 0.000,C 90.000,E1 283.244} C_DIS
LIN {X 0.154,Y -451.747,Z 865.568,A 0.000,B 0.000,C 90.000,E1 282.187} C_DIS
LIN {X -0.152,Y -460.211,Z 865.562,A 0.000,B 0.000,C 90.000,E1 281.186} C_DIS
LIN {X 0.000,Y -468.021,Z 865.556,A 0.000,B 0.000,C 90.000,E1 280.141} C_DIS
LIN {X -0.217,Y -475.204,Z 865.551,A 0.000,B 0.000,C 90.000,E1 279.151} C_DIS
LIN {X -0.226,Y -479.995,Z 865.547,A 0.000,B 0.000,C 90.000,E1 278.398} C_DIS
LIN {X -0.199,Y -484.080,Z 865.542,A 0.000,B 0.000,C 90.000,E1 277.644} C_DIS
LIN {X -0.019,Y -486.381,Z 865.540,A 0.000,B 0.000,C 90.000,E1 277.125} C_DIS
LIN {X 0.178,Y -488.355,Z 865.537,A 0.000,B 0.000,C 90.000,E1 276.606} C_DIS
LIN {X -0.105,Y -490.017,Z 865.534,A 0.000,B 0.000,C 90.000,E1 276.144} C_DIS
LIN {X 0.110,Y -491.333,Z 865.531,A 0.000,B 0.000,C 90.000,E1 275.625} C_DIS
LIN {X -0.156,Y -492.322,Z 865.529,A 0.000,B 0.000,C 90.000,E1 275.163} C_DIS
